// ---- DUTs/IO/Boxes/EPP2339_8DFD1558.TcDUT
{attribute 'GeneratedUsingTerminal: EPP2339-0021-0016'}
{attribute addProperty BoxType "EPP2339-0021-0016"}
{attribute addProperty Description "EPP2339-0021 16 Ch. Dig. Input/Output 24V, 0,5A, M8"}
{attribute addProperty Physics "YY"}
{attribute addProperty Id "Channel_1AT %I*Channel_830843C11Channel_2AT %I*Channel_830843C11Channel_3AT %I*Channel_830843C11Channel_4AT %I*Channel_830843C11Channel_5AT %I*Channel_830843C11Channel_6AT %I*Channel_830843C11Channel_7AT %I*Channel_830843C11Channel_8AT %I*Channel_830843C11Channel_9AT %I*Channel_830843C11Channel_10AT %I*Channel_830843C11Channel_11AT %I*Channel_830843C11Channel_12AT %I*Channel_830843C11Channel_13AT %I*Channel_830843C11Channel_14AT %I*Channel_830843C11Channel_15AT %I*Channel_830843C11Channel_16AT %I*Channel_830843C11Channel_9_1AT %Q*Channel_42CA91F71Channel_10_1AT %Q*Channel_42CA91F71Channel_11_1AT %Q*Channel_42CA91F71Channel_12_1AT %Q*Channel_42CA91F71Channel_13_1AT %Q*Channel_42CA91F71Channel_14_1AT %Q*Channel_42CA91F71Channel_15_1AT %Q*Channel_42CA91F71Channel_16_1AT %Q*Channel_42CA91F71Channel_25AT %Q*Channel_42CA91F71Channel_26AT %Q*Channel_42CA91F71Channel_27AT %Q*Channel_42CA91F71Channel_28AT %Q*Channel_42CA91F71Channel_29AT %Q*Channel_42CA91F71Channel_30AT %Q*Channel_42CA91F71Channel_31AT %Q*Channel_42CA91F71Channel_32AT %Q*Channel_42CA91F71WcStateAT %I*WcState_9091E0EB2InfoDataAT %I*InfoData_6F19DB2B2"}
{attribute addProperty CRC "2382173528"}
{attribute addProperty Size "36"}
TYPE EPP2339_8DFD1558 EXTENDS EtcSlaveBoxBase_77A0E4A7 :
STRUCT
	{attribute addProperty Name "Channel_1"}
	Channel_1 : Channel_830843C1;
	{attribute addProperty Name "Channel_2"}
	Channel_2 : Channel_830843C1;
	{attribute addProperty Name "Channel_3"}
	Channel_3 : Channel_830843C1;
	{attribute addProperty Name "Channel_4"}
	Channel_4 : Channel_830843C1;
	{attribute addProperty Name "Channel_5"}
	Channel_5 : Channel_830843C1;
	{attribute addProperty Name "Channel_6"}
	Channel_6 : Channel_830843C1;
	{attribute addProperty Name "Channel_7"}
	Channel_7 : Channel_830843C1;
	{attribute addProperty Name "Channel_8"}
	Channel_8 : Channel_830843C1;
	{attribute addProperty Name "Channel_9"}
	Channel_9 : Channel_830843C1;
	{attribute addProperty Name "Channel_10"}
	Channel_10 : Channel_830843C1;
	{attribute addProperty Name "Channel_11"}
	Channel_11 : Channel_830843C1;
	{attribute addProperty Name "Channel_12"}
	Channel_12 : Channel_830843C1;
	{attribute addProperty Name "Channel_13"}
	Channel_13 : Channel_830843C1;
	{attribute addProperty Name "Channel_14"}
	Channel_14 : Channel_830843C1;
	{attribute addProperty Name "Channel_15"}
	Channel_15 : Channel_830843C1;
	{attribute addProperty Name "Channel_16"}
	Channel_16 : Channel_830843C1;
	{attribute addProperty Name "Channel_9_1"}
	Channel_9_1 : Channel_42CA91F7;
	{attribute addProperty Name "Channel_10_1"}
	Channel_10_1 : Channel_42CA91F7;
	{attribute addProperty Name "Channel_11_1"}
	Channel_11_1 : Channel_42CA91F7;
	{attribute addProperty Name "Channel_12_1"}
	Channel_12_1 : Channel_42CA91F7;
	{attribute addProperty Name "Channel_13_1"}
	Channel_13_1 : Channel_42CA91F7;
	{attribute addProperty Name "Channel_14_1"}
	Channel_14_1 : Channel_42CA91F7;
	{attribute addProperty Name "Channel_15_1"}
	Channel_15_1 : Channel_42CA91F7;
	{attribute addProperty Name "Channel_16_1"}
	Channel_16_1 : Channel_42CA91F7;
	{attribute addProperty Name "Channel_25"}
	Channel_25 : Channel_42CA91F7;
	{attribute addProperty Name "Channel_26"}
	Channel_26 : Channel_42CA91F7;
	{attribute addProperty Name "Channel_27"}
	Channel_27 : Channel_42CA91F7;
	{attribute addProperty Name "Channel_28"}
	Channel_28 : Channel_42CA91F7;
	{attribute addProperty Name "Channel_29"}
	Channel_29 : Channel_42CA91F7;
	{attribute addProperty Name "Channel_30"}
	Channel_30 : Channel_42CA91F7;
	{attribute addProperty Name "Channel_31"}
	Channel_31 : Channel_42CA91F7;
	{attribute addProperty Name "Channel_32"}
	Channel_32 : Channel_42CA91F7;
	{attribute addProperty Name "WcState"}
	WcState : WcState_9091E0EB;
	{attribute addProperty Name "InfoData"}
	InfoData : InfoData_6F19DB2B;
END_STRUCT
END_TYPE

// ---- DUTs/IO/Boxes/EPP2349_8DFD1558.TcDUT
{attribute 'GeneratedUsingTerminal: EPP2349-0021-0016'}
{attribute addProperty BoxType "EPP2349-0021-0016"}
{attribute addProperty Description "EPP2349-0021 16 Ch. Dig. Input/Output 24V, 10µs, 0,5A, M8"}
{attribute addProperty Physics "YY"}
{attribute addProperty Id "Channel_1AT %I*Channel_830843C11Channel_2AT %I*Channel_830843C11Channel_3AT %I*Channel_830843C11Channel_4AT %I*Channel_830843C11Channel_5AT %I*Channel_830843C11Channel_6AT %I*Channel_830843C11Channel_7AT %I*Channel_830843C11Channel_8AT %I*Channel_830843C11Channel_9AT %I*Channel_830843C11Channel_10AT %I*Channel_830843C11Channel_11AT %I*Channel_830843C11Channel_12AT %I*Channel_830843C11Channel_13AT %I*Channel_830843C11Channel_14AT %I*Channel_830843C11Channel_15AT %I*Channel_830843C11Channel_16AT %I*Channel_830843C11Channel_9_1AT %Q*Channel_42CA91F71Channel_10_1AT %Q*Channel_42CA91F71Channel_11_1AT %Q*Channel_42CA91F71Channel_12_1AT %Q*Channel_42CA91F71Channel_13_1AT %Q*Channel_42CA91F71Channel_14_1AT %Q*Channel_42CA91F71Channel_15_1AT %Q*Channel_42CA91F71Channel_16_1AT %Q*Channel_42CA91F71Channel_25AT %Q*Channel_42CA91F71Channel_26AT %Q*Channel_42CA91F71Channel_27AT %Q*Channel_42CA91F71Channel_28AT %Q*Channel_42CA91F71Channel_29AT %Q*Channel_42CA91F71Channel_30AT %Q*Channel_42CA91F71Channel_31AT %Q*Channel_42CA91F71Channel_32AT %Q*Channel_42CA91F71WcStateAT %I*WcState_9091E0EB2InfoDataAT %I*InfoData_6F19DB2B2"}
{attribute addProperty CRC "2382173528"}
{attribute addProperty Size "36"}
TYPE EPP2349_8DFD1558 EXTENDS EtcSlaveBoxBase_77A0E4A7 :
STRUCT
	{attribute addProperty Name "Channel_1"}
	Channel_1 : Channel_830843C1;
	{attribute addProperty Name "Channel_2"}
	Channel_2 : Channel_830843C1;
	{attribute addProperty Name "Channel_3"}
	Channel_3 : Channel_830843C1;
	{attribute addProperty Name "Channel_4"}
	Channel_4 : Channel_830843C1;
	{attribute addProperty Name "Channel_5"}
	Channel_5 : Channel_830843C1;
	{attribute addProperty Name "Channel_6"}
	Channel_6 : Channel_830843C1;
	{attribute addProperty Name "Channel_7"}
	Channel_7 : Channel_830843C1;
	{attribute addProperty Name "Channel_8"}
	Channel_8 : Channel_830843C1;
	{attribute addProperty Name "Channel_9"}
	Channel_9 : Channel_830843C1;
	{attribute addProperty Name "Channel_10"}
	Channel_10 : Channel_830843C1;
	{attribute addProperty Name "Channel_11"}
	Channel_11 : Channel_830843C1;
	{attribute addProperty Name "Channel_12"}
	Channel_12 : Channel_830843C1;
	{attribute addProperty Name "Channel_13"}
	Channel_13 : Channel_830843C1;
	{attribute addProperty Name "Channel_14"}
	Channel_14 : Channel_830843C1;
	{attribute addProperty Name "Channel_15"}
	Channel_15 : Channel_830843C1;
	{attribute addProperty Name "Channel_16"}
	Channel_16 : Channel_830843C1;
	{attribute addProperty Name "Channel_9_1"}
	Channel_9_1 : Channel_42CA91F7;
	{attribute addProperty Name "Channel_10_1"}
	Channel_10_1 : Channel_42CA91F7;
	{attribute addProperty Name "Channel_11_1"}
	Channel_11_1 : Channel_42CA91F7;
	{attribute addProperty Name "Channel_12_1"}
	Channel_12_1 : Channel_42CA91F7;
	{attribute addProperty Name "Channel_13_1"}
	Channel_13_1 : Channel_42CA91F7;
	{attribute addProperty Name "Channel_14_1"}
	Channel_14_1 : Channel_42CA91F7;
	{attribute addProperty Name "Channel_15_1"}
	Channel_15_1 : Channel_42CA91F7;
	{attribute addProperty Name "Channel_16_1"}
	Channel_16_1 : Channel_42CA91F7;
	{attribute addProperty Name "Channel_25"}
	Channel_25 : Channel_42CA91F7;
	{attribute addProperty Name "Channel_26"}
	Channel_26 : Channel_42CA91F7;
	{attribute addProperty Name "Channel_27"}
	Channel_27 : Channel_42CA91F7;
	{attribute addProperty Name "Channel_28"}
	Channel_28 : Channel_42CA91F7;
	{attribute addProperty Name "Channel_29"}
	Channel_29 : Channel_42CA91F7;
	{attribute addProperty Name "Channel_30"}
	Channel_30 : Channel_42CA91F7;
	{attribute addProperty Name "Channel_31"}
	Channel_31 : Channel_42CA91F7;
	{attribute addProperty Name "Channel_32"}
	Channel_32 : Channel_42CA91F7;
	{attribute addProperty Name "WcState"}
	WcState : WcState_9091E0EB;
	{attribute addProperty Name "InfoData"}
	InfoData : InfoData_6F19DB2B;
END_STRUCT
END_TYPE

// ---- DUTs/IO/Boxes/EP2316_3C060514.TcDUT
{attribute 'GeneratedUsingTerminal: EP2316-0008-0017'}
{attribute addProperty BoxType "EP2316-0008-0017"}
{attribute addProperty Description "EP2316-0008 8 Ch. Dig. In, 10µs, 8Ch. Dig. Out 24V, 0,5A, Diagnostic, D-SUB25"}
{attribute addProperty Physics "YY"}
{attribute addProperty Id "DO_Diag_InputsAT %I*DO_Diag_Inputs_CC4551489DO_Diag_Inputs_1AT %I*DO_Diag_Inputs_212B82C19DO_Inputs_DeviceAT %I*DO_Inputs_Device_AF161A9E4DO_OutputsAT %Q*DO_Outputs_28AC1A9E8DO_Outputs_DeviceAT %Q*DO_Outputs_Device_36A5EF172WcStateAT %I*WcState_9091E0EB2InfoDataAT %I*InfoData_32EB74EA10"}
{attribute addProperty CRC "1007027476"}
{attribute addProperty Size "44"}
TYPE EP2316_3C060514 EXTENDS EtcSlaveBoxBase_77A0E4A7 :
STRUCT
	{attribute addProperty Name "DO_Diag_Inputs"}
	DO_Diag_Inputs : DO_Diag_Inputs_CC455148;
	{attribute addProperty Name "DO_Diag_Inputs_1"}
	DO_Diag_Inputs_1 : DO_Diag_Inputs_212B82C1;
	{attribute addProperty Name "DO_Inputs_Device"}
	DO_Inputs_Device : DO_Inputs_Device_AF161A9E;
	{attribute addProperty Name "DO_Outputs"}
	DO_Outputs : DO_Outputs_28AC1A9E;
	{attribute addProperty Name "DO_Outputs_Device"}
	DO_Outputs_Device : DO_Outputs_Device_36A5EF17;
	{attribute addProperty Name "WcState"}
	WcState : WcState_9091E0EB;
	{attribute addProperty Name "InfoData"}
	InfoData : InfoData_32EB74EA;
END_STRUCT
END_TYPE

// ---- DUTs/IO/Boxes/EP2338_39FFBC52.TcDUT
{attribute 'GeneratedUsingTerminal: EP2338-0001-0016'}
{attribute addProperty BoxType "EP2338-0001-0016"}
{attribute addProperty Description "EP2338-0001 8 Ch. Dig. Input/Output 24V, 0,5A, M8"}
{attribute addProperty Physics "YY"}
{attribute addProperty Id "Channel_1AT %I*Channel_830843C11Channel_2AT %I*Channel_830843C11Channel_3AT %I*Channel_830843C11Channel_4AT %I*Channel_830843C11Channel_5AT %I*Channel_830843C11Channel_6AT %I*Channel_830843C11Channel_7AT %I*Channel_830843C11Channel_8AT %I*Channel_830843C11Channel_1_1AT %Q*Channel_42CA91F71Channel_2_1AT %Q*Channel_42CA91F71Channel_3_1AT %Q*Channel_42CA91F71Channel_4_1AT %Q*Channel_42CA91F71Channel_5_1AT %Q*Channel_42CA91F71Channel_6_1AT %Q*Channel_42CA91F71Channel_7_1AT %Q*Channel_42CA91F71Channel_8_1AT %Q*Channel_42CA91F71WcStateAT %I*WcState_9091E0EB2InfoDataAT %I*InfoData_6F19DB2B2"}
{attribute addProperty CRC "973061202"}
{attribute addProperty Size "20"}
TYPE EP2338_39FFBC52 EXTENDS EtcSlaveBoxBase_77A0E4A7 :
STRUCT
	{attribute addProperty Name "Channel_1"}
	Channel_1 : Channel_830843C1;
	{attribute addProperty Name "Channel_2"}
	Channel_2 : Channel_830843C1;
	{attribute addProperty Name "Channel_3"}
	Channel_3 : Channel_830843C1;
	{attribute addProperty Name "Channel_4"}
	Channel_4 : Channel_830843C1;
	{attribute addProperty Name "Channel_5"}
	Channel_5 : Channel_830843C1;
	{attribute addProperty Name "Channel_6"}
	Channel_6 : Channel_830843C1;
	{attribute addProperty Name "Channel_7"}
	Channel_7 : Channel_830843C1;
	{attribute addProperty Name "Channel_8"}
	Channel_8 : Channel_830843C1;
	{attribute addProperty Name "Channel_1_1"}
	Channel_1_1 : Channel_42CA91F7;
	{attribute addProperty Name "Channel_2_1"}
	Channel_2_1 : Channel_42CA91F7;
	{attribute addProperty Name "Channel_3_1"}
	Channel_3_1 : Channel_42CA91F7;
	{attribute addProperty Name "Channel_4_1"}
	Channel_4_1 : Channel_42CA91F7;
	{attribute addProperty Name "Channel_5_1"}
	Channel_5_1 : Channel_42CA91F7;
	{attribute addProperty Name "Channel_6_1"}
	Channel_6_1 : Channel_42CA91F7;
	{attribute addProperty Name "Channel_7_1"}
	Channel_7_1 : Channel_42CA91F7;
	{attribute addProperty Name "Channel_8_1"}
	Channel_8_1 : Channel_42CA91F7;
	{attribute addProperty Name "WcState"}
	WcState : WcState_9091E0EB;
	{attribute addProperty Name "InfoData"}
	InfoData : InfoData_6F19DB2B;
END_STRUCT
END_TYPE

// ---- DUTs/IO/Boxes/EP2339_C2A6198C.TcDUT
{attribute 'GeneratedUsingTerminal: EP2339-0021-0016'}
{attribute addProperty BoxType "EP2339-0021-0016"}
{attribute addProperty Description "EP2339-0021 16 Ch. Dig. Input/Output 24V, 0,5A, M8"}
{attribute addProperty Physics "YY"}
{attribute addProperty Id "Channel_1AT %I*Channel_830843C11Channel_2AT %I*Channel_830843C11Channel_3AT %I*Channel_830843C11Channel_4AT %I*Channel_830843C11Channel_5AT %I*Channel_830843C11Channel_6AT %I*Channel_830843C11Channel_7AT %I*Channel_830843C11Channel_8AT %I*Channel_830843C11Channel_9AT %I*Channel_830843C11Channel_10AT %I*Channel_830843C11Channel_11AT %I*Channel_830843C11Channel_12AT %I*Channel_830843C11Channel_13AT %I*Channel_830843C11Channel_14AT %I*Channel_830843C11Channel_15AT %I*Channel_830843C11Channel_16AT %I*Channel_830843C11Channel_1_1AT %Q*Channel_42CA91F71Channel_2_1AT %Q*Channel_42CA91F71Channel_3_1AT %Q*Channel_42CA91F71Channel_4_1AT %Q*Channel_42CA91F71Channel_5_1AT %Q*Channel_42CA91F71Channel_6_1AT %Q*Channel_42CA91F71Channel_7_1AT %Q*Channel_42CA91F71Channel_8_1AT %Q*Channel_42CA91F71Channel_9_1AT %Q*Channel_42CA91F71Channel_10_1AT %Q*Channel_42CA91F71Channel_11_1AT %Q*Channel_42CA91F71Channel_12_1AT %Q*Channel_42CA91F71Channel_13_1AT %Q*Channel_42CA91F71Channel_14_1AT %Q*Channel_42CA91F71Channel_15_1AT %Q*Channel_42CA91F71Channel_16_1AT %Q*Channel_42CA91F71WcStateAT %I*WcState_9091E0EB2InfoDataAT %I*InfoData_0A66F0098"}
{attribute addProperty CRC "3265665420"}
{attribute addProperty Size "42"}
TYPE EP2339_C2A6198C EXTENDS EtcSlaveBoxBase_77A0E4A7 :
STRUCT
	{attribute addProperty Name "Channel_1"}
	Channel_1 : Channel_830843C1;
	{attribute addProperty Name "Channel_2"}
	Channel_2 : Channel_830843C1;
	{attribute addProperty Name "Channel_3"}
	Channel_3 : Channel_830843C1;
	{attribute addProperty Name "Channel_4"}
	Channel_4 : Channel_830843C1;
	{attribute addProperty Name "Channel_5"}
	Channel_5 : Channel_830843C1;
	{attribute addProperty Name "Channel_6"}
	Channel_6 : Channel_830843C1;
	{attribute addProperty Name "Channel_7"}
	Channel_7 : Channel_830843C1;
	{attribute addProperty Name "Channel_8"}
	Channel_8 : Channel_830843C1;
	{attribute addProperty Name "Channel_9"}
	Channel_9 : Channel_830843C1;
	{attribute addProperty Name "Channel_10"}
	Channel_10 : Channel_830843C1;
	{attribute addProperty Name "Channel_11"}
	Channel_11 : Channel_830843C1;
	{attribute addProperty Name "Channel_12"}
	Channel_12 : Channel_830843C1;
	{attribute addProperty Name "Channel_13"}
	Channel_13 : Channel_830843C1;
	{attribute addProperty Name "Channel_14"}
	Channel_14 : Channel_830843C1;
	{attribute addProperty Name "Channel_15"}
	Channel_15 : Channel_830843C1;
	{attribute addProperty Name "Channel_16"}
	Channel_16 : Channel_830843C1;
	{attribute addProperty Name "Channel_1_1"}
	Channel_1_1 : Channel_42CA91F7;
	{attribute addProperty Name "Channel_2_1"}
	Channel_2_1 : Channel_42CA91F7;
	{attribute addProperty Name "Channel_3_1"}
	Channel_3_1 : Channel_42CA91F7;
	{attribute addProperty Name "Channel_4_1"}
	Channel_4_1 : Channel_42CA91F7;
	{attribute addProperty Name "Channel_5_1"}
	Channel_5_1 : Channel_42CA91F7;
	{attribute addProperty Name "Channel_6_1"}
	Channel_6_1 : Channel_42CA91F7;
	{attribute addProperty Name "Channel_7_1"}
	Channel_7_1 : Channel_42CA91F7;
	{attribute addProperty Name "Channel_8_1"}
	Channel_8_1 : Channel_42CA91F7;
	{attribute addProperty Name "Channel_9_1"}
	Channel_9_1 : Channel_42CA91F7;
	{attribute addProperty Name "Channel_10_1"}
	Channel_10_1 : Channel_42CA91F7;
	{attribute addProperty Name "Channel_11_1"}
	Channel_11_1 : Channel_42CA91F7;
	{attribute addProperty Name "Channel_12_1"}
	Channel_12_1 : Channel_42CA91F7;
	{attribute addProperty Name "Channel_13_1"}
	Channel_13_1 : Channel_42CA91F7;
	{attribute addProperty Name "Channel_14_1"}
	Channel_14_1 : Channel_42CA91F7;
	{attribute addProperty Name "Channel_15_1"}
	Channel_15_1 : Channel_42CA91F7;
	{attribute addProperty Name "Channel_16_1"}
	Channel_16_1 : Channel_42CA91F7;
	{attribute addProperty Name "WcState"}
	WcState : WcState_9091E0EB;
	{attribute addProperty Name "InfoData"}
	InfoData : InfoData_0A66F009;
END_STRUCT
END_TYPE

// ---- DUTs/IO/Boxes/EP2339_56BCD6FB.TcDUT
{attribute 'GeneratedUsingTerminal: EP2339-0022-0016'}
{attribute addProperty BoxType "EP2339-0022-0016"}
{attribute addProperty Description "EP2339-0022 16 Ch. Dig. Input/Output 24V, 0,5A, M12"}
{attribute addProperty Physics "YY"}
{attribute addProperty Id "Channel_1AT %I*Channel_830843C11Channel_2AT %I*Channel_830843C11Channel_3AT %I*Channel_830843C11Channel_4AT %I*Channel_830843C11Channel_5AT %I*Channel_830843C11Channel_6AT %I*Channel_830843C11Channel_7AT %I*Channel_830843C11Channel_8AT %I*Channel_830843C11Channel_9AT %I*Channel_830843C11Channel_10AT %I*Channel_830843C11Channel_11AT %I*Channel_830843C11Channel_12AT %I*Channel_830843C11Channel_13AT %I*Channel_830843C11Channel_14AT %I*Channel_830843C11Channel_15AT %I*Channel_830843C11Channel_16AT %I*Channel_830843C11Channel_1_1AT %Q*Channel_42CA91F71Channel_2_1AT %Q*Channel_42CA91F71Channel_3_1AT %Q*Channel_42CA91F71Channel_4_1AT %Q*Channel_42CA91F71Channel_5_1AT %Q*Channel_42CA91F71Channel_6_1AT %Q*Channel_42CA91F71Channel_7_1AT %Q*Channel_42CA91F71Channel_8_1AT %Q*Channel_42CA91F71Channel_9_1AT %Q*Channel_42CA91F71Channel_10_1AT %Q*Channel_42CA91F71Channel_11_1AT %Q*Channel_42CA91F71Channel_12_1AT %Q*Channel_42CA91F71Channel_13_1AT %Q*Channel_42CA91F71Channel_14_1AT %Q*Channel_42CA91F71Channel_15_1AT %Q*Channel_42CA91F71Channel_16_1AT %Q*Channel_42CA91F71WcStateAT %I*WcState_9091E0EB2InfoDataAT %I*InfoData_6F19DB2B2"}
{attribute addProperty CRC "1455216379"}
{attribute addProperty Size "36"}
TYPE EP2339_56BCD6FB EXTENDS EtcSlaveBoxBase_77A0E4A7 :
STRUCT
	{attribute addProperty Name "Channel_1"}
	Channel_1 : Channel_830843C1;
	{attribute addProperty Name "Channel_2"}
	Channel_2 : Channel_830843C1;
	{attribute addProperty Name "Channel_3"}
	Channel_3 : Channel_830843C1;
	{attribute addProperty Name "Channel_4"}
	Channel_4 : Channel_830843C1;
	{attribute addProperty Name "Channel_5"}
	Channel_5 : Channel_830843C1;
	{attribute addProperty Name "Channel_6"}
	Channel_6 : Channel_830843C1;
	{attribute addProperty Name "Channel_7"}
	Channel_7 : Channel_830843C1;
	{attribute addProperty Name "Channel_8"}
	Channel_8 : Channel_830843C1;
	{attribute addProperty Name "Channel_9"}
	Channel_9 : Channel_830843C1;
	{attribute addProperty Name "Channel_10"}
	Channel_10 : Channel_830843C1;
	{attribute addProperty Name "Channel_11"}
	Channel_11 : Channel_830843C1;
	{attribute addProperty Name "Channel_12"}
	Channel_12 : Channel_830843C1;
	{attribute addProperty Name "Channel_13"}
	Channel_13 : Channel_830843C1;
	{attribute addProperty Name "Channel_14"}
	Channel_14 : Channel_830843C1;
	{attribute addProperty Name "Channel_15"}
	Channel_15 : Channel_830843C1;
	{attribute addProperty Name "Channel_16"}
	Channel_16 : Channel_830843C1;
	{attribute addProperty Name "Channel_1_1"}
	Channel_1_1 : Channel_42CA91F7;
	{attribute addProperty Name "Channel_2_1"}
	Channel_2_1 : Channel_42CA91F7;
	{attribute addProperty Name "Channel_3_1"}
	Channel_3_1 : Channel_42CA91F7;
	{attribute addProperty Name "Channel_4_1"}
	Channel_4_1 : Channel_42CA91F7;
	{attribute addProperty Name "Channel_5_1"}
	Channel_5_1 : Channel_42CA91F7;
	{attribute addProperty Name "Channel_6_1"}
	Channel_6_1 : Channel_42CA91F7;
	{attribute addProperty Name "Channel_7_1"}
	Channel_7_1 : Channel_42CA91F7;
	{attribute addProperty Name "Channel_8_1"}
	Channel_8_1 : Channel_42CA91F7;
	{attribute addProperty Name "Channel_9_1"}
	Channel_9_1 : Channel_42CA91F7;
	{attribute addProperty Name "Channel_10_1"}
	Channel_10_1 : Channel_42CA91F7;
	{attribute addProperty Name "Channel_11_1"}
	Channel_11_1 : Channel_42CA91F7;
	{attribute addProperty Name "Channel_12_1"}
	Channel_12_1 : Channel_42CA91F7;
	{attribute addProperty Name "Channel_13_1"}
	Channel_13_1 : Channel_42CA91F7;
	{attribute addProperty Name "Channel_14_1"}
	Channel_14_1 : Channel_42CA91F7;
	{attribute addProperty Name "Channel_15_1"}
	Channel_15_1 : Channel_42CA91F7;
	{attribute addProperty Name "Channel_16_1"}
	Channel_16_1 : Channel_42CA91F7;
	{attribute addProperty Name "WcState"}
	WcState : WcState_9091E0EB;
	{attribute addProperty Name "InfoData"}
	InfoData : InfoData_6F19DB2B;
END_STRUCT
END_TYPE

// ---- DUTs/IO/Boxes/EJ5151_905C5FD8.TcDUT
{attribute 'GeneratedUsingTerminal: EJ5151-0000-0016'}
{attribute addProperty BoxType "EJ5151-0000-0016"}
{attribute addProperty Description "EJ5151 1Ch. Inc. Encoder"}
{attribute addProperty Physics "KK"}
{attribute addProperty Id "ENC_InputsAT %I*ENC_Inputs_B353648514ENC_Inputs_1AT %I*ENC_Inputs_24B63C534ENC_OutputsAT %Q*ENC_Outputs_21E2D14D6WcStateAT %I*WcState_9091E0EB2InfoDataAT %I*InfoData_32EB74EA10"}
{attribute addProperty CRC "2421972952"}
{attribute addProperty Size "36"}
TYPE EJ5151_905C5FD8 EXTENDS EtcSlaveTerminalBase_947E5A46 :
STRUCT
	{attribute addProperty Name "ENC_Inputs"}
	ENC_Inputs : ENC_Inputs_B3536485;
	{attribute addProperty Name "ENC_Inputs_1"}
	ENC_Inputs_1 : ENC_Inputs_24B63C53;
	{attribute addProperty Name "ENC_Outputs"}
	ENC_Outputs : ENC_Outputs_21E2D14D;
	{attribute addProperty Name "WcState"}
	WcState : WcState_9091E0EB;
	{attribute addProperty Name "InfoData"}
	InfoData : InfoData_32EB74EA;
END_STRUCT
END_TYPE

// ---- DUTs/IO/Boxes/EL1262_0FA571DE.TcDUT
{attribute 'GeneratedUsingTerminal: EL1262-0000-0002'}
{attribute addProperty BoxType "EL1262-0000-0002"}
{attribute addProperty Description "EL1262 2Ch. Dig. Input 24V, 1µs, DC Oversample"}
{attribute addProperty Physics "KK"}
{attribute addProperty Id "Ch1_CycleCountAT %I*Ch1_CycleCount_9DBE2BC52Ch1_Input_0AT %I*Ch1_Input_FFC4CE241Ch1_Input_1AT %I*Ch1_Input_FFC4CE241Ch1_Input_2AT %I*Ch1_Input_FFC4CE241Ch1_Input_3AT %I*Ch1_Input_FFC4CE241Ch1_Input_4AT %I*Ch1_Input_FFC4CE241Ch1_Input_5AT %I*Ch1_Input_FFC4CE241Ch1_Input_6AT %I*Ch1_Input_FFC4CE241Ch1_Input_7AT %I*Ch1_Input_FFC4CE241Ch1_Input_8AT %I*Ch1_Input_FFC4CE241Ch1_Input_9AT %I*Ch1_Input_FFC4CE241GapAT %I*EMPTY_STRUCTURE0Ch2_CycleCountAT %I*Ch2_CycleCount_976A51B52Ch2_Input_0AT %I*Ch2_Input_78ADA90C1Ch2_Input_1AT %I*Ch2_Input_78ADA90C1Ch2_Input_2AT %I*Ch2_Input_78ADA90C1Ch2_Input_3AT %I*Ch2_Input_78ADA90C1Ch2_Input_4AT %I*Ch2_Input_78ADA90C1Ch2_Input_5AT %I*Ch2_Input_78ADA90C1Ch2_Input_6AT %I*Ch2_Input_78ADA90C1Ch2_Input_7AT %I*Ch2_Input_78ADA90C1Ch2_Input_8AT %I*Ch2_Input_78ADA90C1Ch2_Input_9AT %I*Ch2_Input_78ADA90C1Gap_1AT %I*EMPTY_STRUCTURE0NextSync1TimeAT %I*NextSync1Time_EE185E174WcStateAT %I*WcState_9091E0EB2InfoDataAT %I*InfoData_A7436BC610"}
{attribute addProperty CRC "262500830"}
{attribute addProperty Size "40"}
TYPE EL1262_0FA571DE EXTENDS EtcSlaveTerminalBase_947E5A46 :
STRUCT
	{attribute addProperty Name "Ch1_CycleCount"}
	Ch1_CycleCount : Ch1_CycleCount_9DBE2BC5;
	{attribute addProperty Name "Ch1_Input_0"}
	Ch1_Input_0 : Ch1_Input_FFC4CE24;
	{attribute addProperty Name "Ch1_Input_1"}
	Ch1_Input_1 : Ch1_Input_FFC4CE24;
	{attribute addProperty Name "Ch1_Input_2"}
	Ch1_Input_2 : Ch1_Input_FFC4CE24;
	{attribute addProperty Name "Ch1_Input_3"}
	Ch1_Input_3 : Ch1_Input_FFC4CE24;
	{attribute addProperty Name "Ch1_Input_4"}
	Ch1_Input_4 : Ch1_Input_FFC4CE24;
	{attribute addProperty Name "Ch1_Input_5"}
	Ch1_Input_5 : Ch1_Input_FFC4CE24;
	{attribute addProperty Name "Ch1_Input_6"}
	Ch1_Input_6 : Ch1_Input_FFC4CE24;
	{attribute addProperty Name "Ch1_Input_7"}
	Ch1_Input_7 : Ch1_Input_FFC4CE24;
	{attribute addProperty Name "Ch1_Input_8"}
	Ch1_Input_8 : Ch1_Input_FFC4CE24;
	{attribute addProperty Name "Ch1_Input_9"}
	Ch1_Input_9 : Ch1_Input_FFC4CE24;
	{attribute addProperty Name "Gap"}
	Gap : EMPTY_STRUCTURE;
	{attribute addProperty Name "Ch2_CycleCount"}
	Ch2_CycleCount : Ch2_CycleCount_976A51B5;
	{attribute addProperty Name "Ch2_Input_0"}
	Ch2_Input_0 : Ch2_Input_78ADA90C;
	{attribute addProperty Name "Ch2_Input_1"}
	Ch2_Input_1 : Ch2_Input_78ADA90C;
	{attribute addProperty Name "Ch2_Input_2"}
	Ch2_Input_2 : Ch2_Input_78ADA90C;
	{attribute addProperty Name "Ch2_Input_3"}
	Ch2_Input_3 : Ch2_Input_78ADA90C;
	{attribute addProperty Name "Ch2_Input_4"}
	Ch2_Input_4 : Ch2_Input_78ADA90C;
	{attribute addProperty Name "Ch2_Input_5"}
	Ch2_Input_5 : Ch2_Input_78ADA90C;
	{attribute addProperty Name "Ch2_Input_6"}
	Ch2_Input_6 : Ch2_Input_78ADA90C;
	{attribute addProperty Name "Ch2_Input_7"}
	Ch2_Input_7 : Ch2_Input_78ADA90C;
	{attribute addProperty Name "Ch2_Input_8"}
	Ch2_Input_8 : Ch2_Input_78ADA90C;
	{attribute addProperty Name "Ch2_Input_9"}
	Ch2_Input_9 : Ch2_Input_78ADA90C;
	{attribute addProperty Name "Gap_1"}
	Gap_1 : EMPTY_STRUCTURE;
	{attribute addProperty Name "NextSync1Time"}
	NextSync1Time : NextSync1Time_EE185E17;
	{attribute addProperty Name "WcState"}
	WcState : WcState_9091E0EB;
	{attribute addProperty Name "InfoData"}
	InfoData : InfoData_A7436BC6;
END_STRUCT
END_TYPE

// ---- DUTs/IO/Boxes/EL2262_79C970B1.TcDUT
{attribute 'GeneratedUsingTerminal: EL2262-0000-0001'}
{attribute addProperty BoxType "EL2262-0000-0001"}
{attribute addProperty Description "EL2262 2Ch. Dig. Output 24V, 0.5A, DC Over Sampling"}
{attribute addProperty Physics "KK"}
{attribute addProperty Id "CycCount0AT %Q*CycCount0_2C2338042Sample0_0AT %Q*Sample_0023574C1GapAT %I*EMPTY_STRUCTURE0CycCount1AT %Q*CycCount1_2C2338042Sample1_0AT %Q*Sample_07D5B44A1Gap_1AT %I*EMPTY_STRUCTURE0WcStateAT %I*WcState_0B2B16F91InfoDataAT %I*InfoData_A7436BC610"}
{attribute addProperty CRC "2043244721"}
{attribute addProperty Size "17"}
TYPE EL2262_79C970B1 EXTENDS EtcSlaveTerminalBase_947E5A46 :
STRUCT
	{attribute addProperty Name "CycCount0"}
	CycCount0 : CycCount0_2C233804;
	{attribute addProperty Name "Sample0_0"}
	Sample0_0 : Sample_0023574C;
	{attribute addProperty Name "Gap"}
	Gap : EMPTY_STRUCTURE;
	{attribute addProperty Name "CycCount1"}
	CycCount1 : CycCount1_2C233804;
	{attribute addProperty Name "Sample1_0"}
	Sample1_0 : Sample_07D5B44A;
	{attribute addProperty Name "Gap_1"}
	Gap_1 : EMPTY_STRUCTURE;
	{attribute addProperty Name "WcState"}
	WcState : WcState_0B2B16F9;
	{attribute addProperty Name "InfoData"}
	InfoData : InfoData_A7436BC6;
END_STRUCT
END_TYPE

// ---- DUTs/IO/Boxes/EL2262_147DB6E1.TcDUT
{attribute 'GeneratedUsingTerminal: EL2262-0000-0002'}
{attribute addProperty BoxType "EL2262-0000-0002"}
{attribute addProperty Description "EL2262 2Ch. Dig. Output 24V, 1µs, DC Oversample"}
{attribute addProperty Physics "KK"}
{attribute addProperty Id "CycCount0AT %Q*CycCount0_AF431CE02Sample0_0AT %Q*Sample_0023574C1Sample0_1AT %Q*Sample_0023574C1Sample0_2AT %Q*Sample_0023574C1Sample0_3AT %Q*Sample_0023574C1Sample0_4AT %Q*Sample_0023574C1Sample0_5AT %Q*Sample_0023574C1Sample0_6AT %Q*Sample_0023574C1Sample0_7AT %Q*Sample_0023574C1Sample0_8AT %Q*Sample_0023574C1Sample0_9AT %Q*Sample_0023574C1GapAT %I*EMPTY_STRUCTURE0CycCount1AT %Q*CycCount1_A8B5FFE62Sample1_0AT %Q*Sample_07D5B44A1Sample1_1AT %Q*Sample_07D5B44A1Sample1_2AT %Q*Sample_07D5B44A1Sample1_3AT %Q*Sample_07D5B44A1Sample1_4AT %Q*Sample_07D5B44A1Sample1_5AT %Q*Sample_07D5B44A1Sample1_6AT %Q*Sample_07D5B44A1Sample1_7AT %Q*Sample_07D5B44A1Sample1_8AT %Q*Sample_07D5B44A1Sample1_9AT %Q*Sample_07D5B44A1Gap_1AT %I*EMPTY_STRUCTURE0WcStateAT %I*WcState_0B2B16F91InfoDataAT %I*InfoData_A7436BC610"}
{attribute addProperty CRC "343783137"}
{attribute addProperty Size "35"}
TYPE EL2262_147DB6E1 EXTENDS EtcSlaveTerminalBase_947E5A46 :
STRUCT
	{attribute addProperty Name "CycCount0"}
	CycCount0 : CycCount0_AF431CE0;
	{attribute addProperty Name "Sample0_0"}
	Sample0_0 : Sample_0023574C;
	{attribute addProperty Name "Sample0_1"}
	Sample0_1 : Sample_0023574C;
	{attribute addProperty Name "Sample0_2"}
	Sample0_2 : Sample_0023574C;
	{attribute addProperty Name "Sample0_3"}
	Sample0_3 : Sample_0023574C;
	{attribute addProperty Name "Sample0_4"}
	Sample0_4 : Sample_0023574C;
	{attribute addProperty Name "Sample0_5"}
	Sample0_5 : Sample_0023574C;
	{attribute addProperty Name "Sample0_6"}
	Sample0_6 : Sample_0023574C;
	{attribute addProperty Name "Sample0_7"}
	Sample0_7 : Sample_0023574C;
	{attribute addProperty Name "Sample0_8"}
	Sample0_8 : Sample_0023574C;
	{attribute addProperty Name "Sample0_9"}
	Sample0_9 : Sample_0023574C;
	{attribute addProperty Name "Gap"}
	Gap : EMPTY_STRUCTURE;
	{attribute addProperty Name "CycCount1"}
	CycCount1 : CycCount1_A8B5FFE6;
	{attribute addProperty Name "Sample1_0"}
	Sample1_0 : Sample_07D5B44A;
	{attribute addProperty Name "Sample1_1"}
	Sample1_1 : Sample_07D5B44A;
	{attribute addProperty Name "Sample1_2"}
	Sample1_2 : Sample_07D5B44A;
	{attribute addProperty Name "Sample1_3"}
	Sample1_3 : Sample_07D5B44A;
	{attribute addProperty Name "Sample1_4"}
	Sample1_4 : Sample_07D5B44A;
	{attribute addProperty Name "Sample1_5"}
	Sample1_5 : Sample_07D5B44A;
	{attribute addProperty Name "Sample1_6"}
	Sample1_6 : Sample_07D5B44A;
	{attribute addProperty Name "Sample1_7"}
	Sample1_7 : Sample_07D5B44A;
	{attribute addProperty Name "Sample1_8"}
	Sample1_8 : Sample_07D5B44A;
	{attribute addProperty Name "Sample1_9"}
	Sample1_9 : Sample_07D5B44A;
	{attribute addProperty Name "Gap_1"}
	Gap_1 : EMPTY_STRUCTURE;
	{attribute addProperty Name "WcState"}
	WcState : WcState_0B2B16F9;
	{attribute addProperty Name "InfoData"}
	InfoData : InfoData_A7436BC6;
END_STRUCT
END_TYPE

// ---- DUTs/IO/Boxes/EL2262_9619875D.TcDUT
{attribute 'GeneratedUsingTerminal: EL2262-0000-0004'}
{attribute addProperty BoxType "EL2262-0000-0004"}
{attribute addProperty Description "EL2262 2Ch. Dig. Output 24V, 1µs, DC Oversample"}
{attribute addProperty Physics "KK"}
{attribute addProperty Id "StartTimeNextOutputAT %I*StartTimeNextOutput_228767F44CycCount0AT %Q*CycCount0_AF431CE02Sample0_0AT %Q*Sample_0023574C1Sample0_1AT %Q*Sample_0023574C1Sample0_2AT %Q*Sample_0023574C1Sample0_3AT %Q*Sample_0023574C1Sample0_4AT %Q*Sample_0023574C1Sample0_5AT %Q*Sample_0023574C1Sample0_6AT %Q*Sample_0023574C1Sample0_7AT %Q*Sample_0023574C1Sample0_8AT %Q*Sample_0023574C1Sample0_9AT %Q*Sample_0023574C1GapAT %I*EMPTY_STRUCTURE0CycCount1AT %Q*CycCount1_A8B5FFE62Sample1_0AT %Q*Sample_07D5B44A1Sample1_1AT %Q*Sample_07D5B44A1Sample1_2AT %Q*Sample_07D5B44A1Sample1_3AT %Q*Sample_07D5B44A1Sample1_4AT %Q*Sample_07D5B44A1Sample1_5AT %Q*Sample_07D5B44A1Sample1_6AT %Q*Sample_07D5B44A1Sample1_7AT %Q*Sample_07D5B44A1Sample1_8AT %Q*Sample_07D5B44A1Sample1_9AT %Q*Sample_07D5B44A1Gap_1AT %I*EMPTY_STRUCTURE0WcStateAT %I*WcState_9091E0EB2InfoDataAT %I*InfoData_A7436BC610"}
{attribute addProperty CRC "2518255453"}
{attribute addProperty Size "40"}
TYPE EL2262_9619875D EXTENDS EtcSlaveTerminalBase_947E5A46 :
STRUCT
	{attribute addProperty Name "StartTimeNextOutput"}
	StartTimeNextOutput : StartTimeNextOutput_228767F4;
	{attribute addProperty Name "CycCount0"}
	CycCount0 : CycCount0_AF431CE0;
	{attribute addProperty Name "Sample0_0"}
	Sample0_0 : Sample_0023574C;
	{attribute addProperty Name "Sample0_1"}
	Sample0_1 : Sample_0023574C;
	{attribute addProperty Name "Sample0_2"}
	Sample0_2 : Sample_0023574C;
	{attribute addProperty Name "Sample0_3"}
	Sample0_3 : Sample_0023574C;
	{attribute addProperty Name "Sample0_4"}
	Sample0_4 : Sample_0023574C;
	{attribute addProperty Name "Sample0_5"}
	Sample0_5 : Sample_0023574C;
	{attribute addProperty Name "Sample0_6"}
	Sample0_6 : Sample_0023574C;
	{attribute addProperty Name "Sample0_7"}
	Sample0_7 : Sample_0023574C;
	{attribute addProperty Name "Sample0_8"}
	Sample0_8 : Sample_0023574C;
	{attribute addProperty Name "Sample0_9"}
	Sample0_9 : Sample_0023574C;
	{attribute addProperty Name "Gap"}
	Gap : EMPTY_STRUCTURE;
	{attribute addProperty Name "CycCount1"}
	CycCount1 : CycCount1_A8B5FFE6;
	{attribute addProperty Name "Sample1_0"}
	Sample1_0 : Sample_07D5B44A;
	{attribute addProperty Name "Sample1_1"}
	Sample1_1 : Sample_07D5B44A;
	{attribute addProperty Name "Sample1_2"}
	Sample1_2 : Sample_07D5B44A;
	{attribute addProperty Name "Sample1_3"}
	Sample1_3 : Sample_07D5B44A;
	{attribute addProperty Name "Sample1_4"}
	Sample1_4 : Sample_07D5B44A;
	{attribute addProperty Name "Sample1_5"}
	Sample1_5 : Sample_07D5B44A;
	{attribute addProperty Name "Sample1_6"}
	Sample1_6 : Sample_07D5B44A;
	{attribute addProperty Name "Sample1_7"}
	Sample1_7 : Sample_07D5B44A;
	{attribute addProperty Name "Sample1_8"}
	Sample1_8 : Sample_07D5B44A;
	{attribute addProperty Name "Sample1_9"}
	Sample1_9 : Sample_07D5B44A;
	{attribute addProperty Name "Gap_1"}
	Gap_1 : EMPTY_STRUCTURE;
	{attribute addProperty Name "WcState"}
	WcState : WcState_9091E0EB;
	{attribute addProperty Name "InfoData"}
	InfoData : InfoData_A7436BC6;
END_STRUCT
END_TYPE

// ---- DUTs/IO/Boxes/EL3681_02A14E64.TcDUT
{attribute 'GeneratedUsingTerminal: EL3681-0000-0017'}
{attribute addProperty BoxType "EL3681-0000-0017"}
{attribute addProperty Description "EL3681 digital multimeter terminal"}
{attribute addProperty Physics "KK"}
{attribute addProperty Id "SAI_InputsAT %I*SAI_Inputs_3A838E1114SAI_RangeAT %I*SAI_Range_C3200E782SAI_Range_1AT %Q*SAI_Range_3710D7473WcStateAT %I*WcState_9091E0EB2InfoDataAT %I*InfoData_32EB74EA10"}
{attribute addProperty CRC "44125796"}
{attribute addProperty Size "31"}
TYPE EL3681_02A14E64 EXTENDS EtcSlaveTerminalBase_947E5A46 :
STRUCT
	{attribute addProperty Name "SAI_Inputs"}
	SAI_Inputs : SAI_Inputs_3A838E11;
	{attribute addProperty Name "SAI_Range"}
	SAI_Range : SAI_Range_C3200E78;
	{attribute addProperty Name "SAI_Range_1"}
	SAI_Range_1 : SAI_Range_3710D747;
	{attribute addProperty Name "WcState"}
	WcState : WcState_9091E0EB;
	{attribute addProperty Name "InfoData"}
	InfoData : InfoData_32EB74EA;
END_STRUCT
END_TYPE

// ---- DUTs/IO/Boxes/EL3681_0095B62C.TcDUT
{attribute 'GeneratedUsingTerminal: EL3681-0000-0018'}
{attribute addProperty BoxType "EL3681-0000-0018"}
{attribute addProperty Description "EL3681 Digital multimeter terminal"}
{attribute addProperty Physics "KK"}
{attribute addProperty Id "SAI_InputsAT %I*SAI_Inputs_84B29FE914SAI_RangeAT %I*SAI_Range_BDBF6DA92SAI_Range_1AT %Q*SAI_Range_2A187FC54WcStateAT %I*WcState_9091E0EB2InfoDataAT %I*InfoData_32EB74EA10"}
{attribute addProperty CRC "9811500"}
{attribute addProperty Size "32"}
TYPE EL3681_0095B62C EXTENDS EtcSlaveTerminalBase_947E5A46 :
STRUCT
	{attribute addProperty Name "SAI_Inputs"}
	SAI_Inputs : SAI_Inputs_84B29FE9;
	{attribute addProperty Name "SAI_Range"}
	SAI_Range : SAI_Range_BDBF6DA9;
	{attribute addProperty Name "SAI_Range_1"}
	SAI_Range_1 : SAI_Range_2A187FC5;
	{attribute addProperty Name "WcState"}
	WcState : WcState_9091E0EB;
	{attribute addProperty Name "InfoData"}
	InfoData : InfoData_32EB74EA;
END_STRUCT
END_TYPE

// ---- DUTs/IO/Boxes/EL5101_127DF9F1.TcDUT
{attribute 'GeneratedUsingTerminal: EL5101--0000'}
{attribute addProperty BoxType "EL5101--0000"}
{attribute addProperty Description "EL5101 1Ch. Encoder 5V"}
{attribute addProperty Physics "KK"}
{attribute addProperty Id "Channel_1AT %I*Channel_B90637B95Channel_1_1AT %Q*Channel_C6781B153WcStateAT %I*WcState_9091E0EB2InfoDataAT %I*InfoData_32EB74EA10"}
{attribute addProperty CRC "310245873"}
{attribute addProperty Size "20"}
TYPE EL5101_127DF9F1 EXTENDS EtcSlaveTerminalBase_947E5A46 :
STRUCT
	{attribute addProperty Name "Channel_1"}
	Channel_1 : Channel_B90637B9;
	{attribute addProperty Name "Channel_1_1"}
	Channel_1_1 : Channel_C6781B15;
	{attribute addProperty Name "WcState"}
	WcState : WcState_9091E0EB;
	{attribute addProperty Name "InfoData"}
	InfoData : InfoData_32EB74EA;
END_STRUCT
END_TYPE

// ---- DUTs/IO/Boxes/EL5151_84FDBA5C.TcDUT
{attribute 'GeneratedUsingTerminal: EL5151-0000-0016'}
{attribute addProperty BoxType "EL5151-0000-0016"}
{attribute addProperty Description "EL5151 1Ch. Inc. Encoder"}
{attribute addProperty Physics "KK"}
{attribute addProperty Id "ENC_InputsAT %I*ENC_Inputs_3399C5AA16ENC_Inputs_1AT %I*ENC_Inputs_24B63C534ENC_OutputsAT %Q*ENC_Outputs_2E45048F8WcStateAT %I*WcState_9091E0EB2InfoDataAT %I*InfoData_32EB74EA10"}
{attribute addProperty CRC "2231220828"}
{attribute addProperty Size "40"}
TYPE EL5151_84FDBA5C EXTENDS EtcSlaveTerminalBase_947E5A46 :
STRUCT
	{attribute addProperty Name "ENC_Inputs"}
	ENC_Inputs : ENC_Inputs_3399C5AA;
	{attribute addProperty Name "ENC_Inputs_1"}
	ENC_Inputs_1 : ENC_Inputs_24B63C53;
	{attribute addProperty Name "ENC_Outputs"}
	ENC_Outputs : ENC_Outputs_2E45048F;
	{attribute addProperty Name "WcState"}
	WcState : WcState_9091E0EB;
	{attribute addProperty Name "InfoData"}
	InfoData : InfoData_32EB74EA;
END_STRUCT
END_TYPE

// ---- DUTs/IO/Boxes/EL5151_93354628.TcDUT
{attribute 'GeneratedUsingTerminal: EL5151-0000-0017'}
{attribute addProperty BoxType "EL5151-0000-0017"}
{attribute addProperty Description "EL5151 1Ch. Inc. Encoder"}
{attribute addProperty Physics "KK"}
{attribute addProperty Id "ENC_InputsAT %I*ENC_Inputs_561E041F18ENC_Inputs_1AT %I*ENC_Inputs_24B63C534ENC_OutputsAT %Q*ENC_Outputs_2E45048F8WcStateAT %I*WcState_9091E0EB2InfoDataAT %I*InfoData_32EB74EA10"}
{attribute addProperty CRC "2469742120"}
{attribute addProperty Size "42"}
TYPE EL5151_93354628 EXTENDS EtcSlaveTerminalBase_947E5A46 :
STRUCT
	{attribute addProperty Name "ENC_Inputs"}
	ENC_Inputs : ENC_Inputs_561E041F;
	{attribute addProperty Name "ENC_Inputs_1"}
	ENC_Inputs_1 : ENC_Inputs_24B63C53;
	{attribute addProperty Name "ENC_Outputs"}
	ENC_Outputs : ENC_Outputs_2E45048F;
	{attribute addProperty Name "WcState"}
	WcState : WcState_9091E0EB;
	{attribute addProperty Name "InfoData"}
	InfoData : InfoData_32EB74EA;
END_STRUCT
END_TYPE

// ---- DUTs/IO/Boxes/EL5151_905C5FD8.TcDUT
{attribute 'GeneratedUsingTerminal: EL5151-0000-0020'}
{attribute addProperty BoxType "EL5151-0000-0020"}
{attribute addProperty Description "EL5151 1Ch. Inc. Encoder"}
{attribute addProperty Physics "KK"}
{attribute addProperty Id "ENC_InputsAT %I*ENC_Inputs_B353648514ENC_Inputs_1AT %I*ENC_Inputs_24B63C534ENC_OutputsAT %Q*ENC_Outputs_21E2D14D6WcStateAT %I*WcState_9091E0EB2InfoDataAT %I*InfoData_32EB74EA10"}
{attribute addProperty CRC "2421972952"}
{attribute addProperty Size "36"}
TYPE EL5151_905C5FD8 EXTENDS EtcSlaveTerminalBase_947E5A46 :
STRUCT
	{attribute addProperty Name "ENC_Inputs"}
	ENC_Inputs : ENC_Inputs_B3536485;
	{attribute addProperty Name "ENC_Inputs_1"}
	ENC_Inputs_1 : ENC_Inputs_24B63C53;
	{attribute addProperty Name "ENC_Outputs"}
	ENC_Outputs : ENC_Outputs_21E2D14D;
	{attribute addProperty Name "WcState"}
	WcState : WcState_9091E0EB;
	{attribute addProperty Name "InfoData"}
	InfoData : InfoData_32EB74EA;
END_STRUCT
END_TYPE

// ---- DUTs/IO/Boxes/EL5151_4D0E77FC.TcDUT
{attribute 'GeneratedUsingTerminal: EL5151-0080-0016'}
{attribute addProperty BoxType "EL5151-0080-0016"}
{attribute addProperty Description "EL5151-0080 1Ch. Inc. Encoder (250kHz)"}
{attribute addProperty Physics "KK"}
{attribute addProperty Id "ENC_InputsAT %I*ENC_Inputs_F139456B14ENC_Inputs_1AT %I*ENC_Inputs_24B63C534ENC_OutputsAT %Q*ENC_Outputs_6FDDC6696WcStateAT %I*WcState_9091E0EB2InfoDataAT %I*InfoData_32EB74EA10"}
{attribute addProperty CRC "1292793852"}
{attribute addProperty Size "36"}
TYPE EL5151_4D0E77FC EXTENDS EtcSlaveTerminalBase_947E5A46 :
STRUCT
	{attribute addProperty Name "ENC_Inputs"}
	ENC_Inputs : ENC_Inputs_F139456B;
	{attribute addProperty Name "ENC_Inputs_1"}
	ENC_Inputs_1 : ENC_Inputs_24B63C53;
	{attribute addProperty Name "ENC_Outputs"}
	ENC_Outputs : ENC_Outputs_6FDDC669;
	{attribute addProperty Name "WcState"}
	WcState : WcState_9091E0EB;
	{attribute addProperty Name "InfoData"}
	InfoData : InfoData_32EB74EA;
END_STRUCT
END_TYPE

// ---- DUTs/IO/Boxes/EL3773_D0D76902.TcDUT
{attribute 'GeneratedUsingTerminal: EL3773-0000-0016'}
{attribute addProperty BoxType "EL3773-0000-0016"}
{attribute addProperty Description "EL3773 3 Ch. Power Monitoring, Oversample"}
{attribute addProperty Physics "KK"}
{attribute addProperty Id "L1_Voltage_StatusAT %I*L1_Voltage_Status_784F03AD8L1_Voltage_SamplesAT %I*L1_Voltage_Samples_ED678DEE20L1_Current_SamplesAT %I*L1_Current_Samples_89E078188L1_Current_Samples_1AT %I*L1_Current_Samples_3209B12F20L2_Voltage_StatusAT %I*L2_Voltage_Status_0626A0108L2_Voltage_SamplesAT %I*L2_Voltage_Samples_D91109BE20L2_Current_StatusAT %I*L2_Current_Status_F789DBA58L2_Current_SamplesAT %I*L2_Current_Samples_067F357F20L3_Voltage_StatusAT %I*L3_Voltage_Status_2C01C17B8L3_Voltage_SamplesAT %I*L3_Voltage_Samples_CAC3758E20L3_Current_StatusAT %I*L3_Current_Status_DDAEBACE8L3_Current_SamplesAT %I*L3_Current_Samples_15AD494F20AI_Timestamp_NextSync1TimeAT %I*AI_Timestamp_NextSync1Time_9AFDC2758AI_CycleCountAT %I*AI_CycleCount_B1A935A22WcStateAT %I*WcState_9091E0EB2InfoDataAT %I*InfoData_BEF6B88E18"}
{attribute addProperty CRC "3503778050"}
{attribute addProperty Size "198"}
TYPE EL3773_D0D76902 EXTENDS EtcSlaveTerminalBase_947E5A46 :
STRUCT
	{attribute addProperty Name "L1_Voltage_Status"}
	L1_Voltage_Status : L1_Voltage_Status_784F03AD;
	{attribute addProperty Name "L1_Voltage_Samples"}
	L1_Voltage_Samples : L1_Voltage_Samples_ED678DEE;
	{attribute addProperty Name "L1_Current_Samples"}
	L1_Current_Samples : L1_Current_Samples_89E07818;
	{attribute addProperty Name "L1_Current_Samples_1"}
	L1_Current_Samples_1 : L1_Current_Samples_3209B12F;
	{attribute addProperty Name "L2_Voltage_Status"}
	L2_Voltage_Status : L2_Voltage_Status_0626A010;
	{attribute addProperty Name "L2_Voltage_Samples"}
	L2_Voltage_Samples : L2_Voltage_Samples_D91109BE;
	{attribute addProperty Name "L2_Current_Status"}
	L2_Current_Status : L2_Current_Status_F789DBA5;
	{attribute addProperty Name "L2_Current_Samples"}
	L2_Current_Samples : L2_Current_Samples_067F357F;
	{attribute addProperty Name "L3_Voltage_Status"}
	L3_Voltage_Status : L3_Voltage_Status_2C01C17B;
	{attribute addProperty Name "L3_Voltage_Samples"}
	L3_Voltage_Samples : L3_Voltage_Samples_CAC3758E;
	{attribute addProperty Name "L3_Current_Status"}
	L3_Current_Status : L3_Current_Status_DDAEBACE;
	{attribute addProperty Name "L3_Current_Samples"}
	L3_Current_Samples : L3_Current_Samples_15AD494F;
	{attribute addProperty Name "AI_Timestamp_NextSync1Time"}
	AI_Timestamp_NextSync1Time : AI_Timestamp_NextSync1Time_9AFDC275;
	{attribute addProperty Name "AI_CycleCount"}
	AI_CycleCount : AI_CycleCount_B1A935A2;
	{attribute addProperty Name "WcState"}
	WcState : WcState_9091E0EB;
	{attribute addProperty Name "InfoData"}
	InfoData : InfoData_BEF6B88E;
END_STRUCT
END_TYPE

// ---- DUTs/IO/Boxes/EM7004_866015E1.TcDUT
{attribute 'GeneratedUsingTerminal: EM7004-0000-9995'}
{attribute addProperty BoxType "EM7004-0000-9995"}
{attribute addProperty Description "EM7004 4-Axis Interface Unit"}
{attribute addProperty Physics "KK"}
{attribute addProperty Id "DigitalAT %I*Digital_BD004D6F16Encoder_Channel_1AT %I*Encoder_Channel_2E4EA2136Encoder_Channel_2AT %I*Encoder_Channel_2E4EA2136Encoder_Channel_3AT %I*Encoder_Channel_2E4EA2136Encoder_Channel_4AT %I*Encoder_Channel_2E4EA2136Digital_1AT %Q*Digital_A7E1DFAB16Analog_Channel_1AT %Q*Analog_Channel_5F9B7EA62Analog_Channel_2AT %Q*Analog_Channel_5F9B7EA62Analog_Channel_3AT %Q*Analog_Channel_5F9B7EA62Analog_Channel_4AT %Q*Analog_Channel_5F9B7EA62Encoder_Channel_1_1AT %Q*Encoder_Channel_B7999E144Encoder_Channel_2_1AT %Q*Encoder_Channel_B7999E144Encoder_Channel_3_1AT %Q*Encoder_Channel_B7999E144Encoder_Channel_4_1AT %Q*Encoder_Channel_B7999E144WcStateAT %I*WcState_9091E0EB2InfoDataAT %I*InfoData_32EB74EA10"}
{attribute addProperty CRC "2254444001"}
{attribute addProperty Size "92"}
TYPE EM7004_866015E1 EXTENDS EtcSlaveTerminalBase_947E5A46 :
STRUCT
	{attribute addProperty Name "Digital"}
	Digital : Digital_BD004D6F;
	{attribute addProperty Name "Encoder_Channel_1"}
	Encoder_Channel_1 : Encoder_Channel_2E4EA213;
	{attribute addProperty Name "Encoder_Channel_2"}
	Encoder_Channel_2 : Encoder_Channel_2E4EA213;
	{attribute addProperty Name "Encoder_Channel_3"}
	Encoder_Channel_3 : Encoder_Channel_2E4EA213;
	{attribute addProperty Name "Encoder_Channel_4"}
	Encoder_Channel_4 : Encoder_Channel_2E4EA213;
	{attribute addProperty Name "Digital_1"}
	Digital_1 : Digital_A7E1DFAB;
	{attribute addProperty Name "Analog_Channel_1"}
	Analog_Channel_1 : Analog_Channel_5F9B7EA6;
	{attribute addProperty Name "Analog_Channel_2"}
	Analog_Channel_2 : Analog_Channel_5F9B7EA6;
	{attribute addProperty Name "Analog_Channel_3"}
	Analog_Channel_3 : Analog_Channel_5F9B7EA6;
	{attribute addProperty Name "Analog_Channel_4"}
	Analog_Channel_4 : Analog_Channel_5F9B7EA6;
	{attribute addProperty Name "Encoder_Channel_1_1"}
	Encoder_Channel_1_1 : Encoder_Channel_B7999E14;
	{attribute addProperty Name "Encoder_Channel_2_1"}
	Encoder_Channel_2_1 : Encoder_Channel_B7999E14;
	{attribute addProperty Name "Encoder_Channel_3_1"}
	Encoder_Channel_3_1 : Encoder_Channel_B7999E14;
	{attribute addProperty Name "Encoder_Channel_4_1"}
	Encoder_Channel_4_1 : Encoder_Channel_B7999E14;
	{attribute addProperty Name "WcState"}
	WcState : WcState_9091E0EB;
	{attribute addProperty Name "InfoData"}
	InfoData : InfoData_32EB74EA;
END_STRUCT
END_TYPE

// ---- DUTs/IO/Boxes/AX8108_8297A621.TcDUT
{attribute 'GeneratedUsingTerminal: AX8108-0100-0101-0101'}
{attribute addProperty BoxType "AX8108-0100-0101-0101"}
{attribute addProperty Description "AX8108-0100-0101"}
{attribute addProperty Physics "KK"}
{attribute addProperty Id "DeviceDevice_6E2575772Device_SafetyDevice_Safety_C21945A160Ch_ACh_A_1FF86D8522WcStateAT %I*WcState_B516A2644InfoDataAT %I*InfoData_358A59CF25"}
{attribute addProperty CRC "2190976545"}
{attribute addProperty Size "113"}
TYPE AX8108_8297A621 EXTENDS EtcSlaveTerminalBase_947E5A46 :
STRUCT
	{attribute addProperty Name "Device"}
	Device : Device_6E257577;
	{attribute addProperty Name "Device_Safety"}
	Device_Safety : Device_Safety_C21945A1;
	{attribute addProperty Name "Ch_A"}
	Ch_A : Ch_A_1FF86D85;
	{attribute addProperty Name "WcState"}
	WcState : WcState_B516A264;
	{attribute addProperty Name "InfoData"}
	InfoData : InfoData_358A59CF;
END_STRUCT
END_TYPE

// ---- DUTs/IO/Boxes/AX8108_F7A82895.TcDUT
{attribute 'GeneratedUsingTerminal: AX8108-0100-0102-0102'}
{attribute addProperty BoxType "AX8108-0100-0102-0102"}
{attribute addProperty Description "AX8108-0100-0102"}
{attribute addProperty Physics "KK"}
{attribute addProperty Id "DeviceDevice_6E2575772Device_SafetyDevice_Safety_C21945A160Ch_ACh_A_D18C6F1622WcStateAT %I*WcState_B516A2644InfoDataAT %I*InfoData_358A59CF25"}
{attribute addProperty CRC "4154992789"}
{attribute addProperty Size "113"}
TYPE AX8108_F7A82895 EXTENDS EtcSlaveTerminalBase_947E5A46 :
STRUCT
	{attribute addProperty Name "Device"}
	Device : Device_6E257577;
	{attribute addProperty Name "Device_Safety"}
	Device_Safety : Device_Safety_C21945A1;
	{attribute addProperty Name "Ch_A"}
	Ch_A : Ch_A_D18C6F16;
	{attribute addProperty Name "WcState"}
	WcState : WcState_B516A264;
	{attribute addProperty Name "InfoData"}
	InfoData : InfoData_358A59CF;
END_STRUCT
END_TYPE

// ---- DUTs/IO/Boxes/AX8118_8297A621.TcDUT
{attribute 'GeneratedUsingTerminal: AX8118-0100-0101-0101'}
{attribute addProperty BoxType "AX8118-0100-0101-0101"}
{attribute addProperty Description "AX8118-0100-0101"}
{attribute addProperty Physics "KK"}
{attribute addProperty Id "DeviceDevice_6E2575772Device_SafetyDevice_Safety_C21945A160Ch_ACh_A_1FF86D8522WcStateAT %I*WcState_B516A2644InfoDataAT %I*InfoData_358A59CF25"}
{attribute addProperty CRC "2190976545"}
{attribute addProperty Size "113"}
TYPE AX8118_8297A621 EXTENDS EtcSlaveTerminalBase_947E5A46 :
STRUCT
	{attribute addProperty Name "Device"}
	Device : Device_6E257577;
	{attribute addProperty Name "Device_Safety"}
	Device_Safety : Device_Safety_C21945A1;
	{attribute addProperty Name "Ch_A"}
	Ch_A : Ch_A_1FF86D85;
	{attribute addProperty Name "WcState"}
	WcState : WcState_B516A264;
	{attribute addProperty Name "InfoData"}
	InfoData : InfoData_358A59CF;
END_STRUCT
END_TYPE

// ---- DUTs/IO/Boxes/AX8118_F7A82895.TcDUT
{attribute 'GeneratedUsingTerminal: AX8118-0100-0102-0102'}
{attribute addProperty BoxType "AX8118-0100-0102-0102"}
{attribute addProperty Description "AX8118-0100-0102"}
{attribute addProperty Physics "KK"}
{attribute addProperty Id "DeviceDevice_6E2575772Device_SafetyDevice_Safety_C21945A160Ch_ACh_A_D18C6F1622WcStateAT %I*WcState_B516A2644InfoDataAT %I*InfoData_358A59CF25"}
{attribute addProperty CRC "4154992789"}
{attribute addProperty Size "113"}
TYPE AX8118_F7A82895 EXTENDS EtcSlaveTerminalBase_947E5A46 :
STRUCT
	{attribute addProperty Name "Device"}
	Device : Device_6E257577;
	{attribute addProperty Name "Device_Safety"}
	Device_Safety : Device_Safety_C21945A1;
	{attribute addProperty Name "Ch_A"}
	Ch_A : Ch_A_D18C6F16;
	{attribute addProperty Name "WcState"}
	WcState : WcState_B516A264;
	{attribute addProperty Name "InfoData"}
	InfoData : InfoData_358A59CF;
END_STRUCT
END_TYPE

// ---- DUTs/IO/Boxes/AX8206_63F473B4.TcDUT
{attribute 'GeneratedUsingTerminal: AX8206-0100-0101-0101'}
{attribute addProperty BoxType "AX8206-0100-0101-0101"}
{attribute addProperty Description "AX8206-0100-0101"}
{attribute addProperty Physics "KK"}
{attribute addProperty Id "DeviceDevice_6E2575772Device_SafetyDevice_Safety_C21945A160Ch_ACh_A_1FF86D8522Ch_BCh_B_5E084BAA22WcStateAT %I*WcState_B516A2644InfoDataAT %I*InfoData_386C00A526"}
{attribute addProperty CRC "1676964788"}
{attribute addProperty Size "136"}
TYPE AX8206_63F473B4 EXTENDS EtcSlaveTerminalBase_947E5A46 :
STRUCT
	{attribute addProperty Name "Device"}
	Device : Device_6E257577;
	{attribute addProperty Name "Device_Safety"}
	Device_Safety : Device_Safety_C21945A1;
	{attribute addProperty Name "Ch_A"}
	Ch_A : Ch_A_1FF86D85;
	{attribute addProperty Name "Ch_B"}
	Ch_B : Ch_B_5E084BAA;
	{attribute addProperty Name "WcState"}
	WcState : WcState_B516A264;
	{attribute addProperty Name "InfoData"}
	InfoData : InfoData_386C00A5;
END_STRUCT
END_TYPE

// ---- DUTs/IO/Boxes/AX8206_FA9FF81E.TcDUT
{attribute 'GeneratedUsingTerminal: AX8206-0100-0102-0102'}
{attribute addProperty BoxType "AX8206-0100-0102-0102"}
{attribute addProperty Description "AX8206-0100-0102"}
{attribute addProperty Physics "KK"}
{attribute addProperty Id "DeviceDevice_6E2575772Device_SafetyDevice_Safety_C21945A160Ch_ACh_A_D18C6F1622Ch_BCh_B_647F9A0C22WcStateAT %I*WcState_B516A2644InfoDataAT %I*InfoData_386C00A526"}
{attribute addProperty CRC "4204787742"}
{attribute addProperty Size "136"}
TYPE AX8206_FA9FF81E EXTENDS EtcSlaveTerminalBase_947E5A46 :
STRUCT
	{attribute addProperty Name "Device"}
	Device : Device_6E257577;
	{attribute addProperty Name "Device_Safety"}
	Device_Safety : Device_Safety_C21945A1;
	{attribute addProperty Name "Ch_A"}
	Ch_A : Ch_A_D18C6F16;
	{attribute addProperty Name "Ch_B"}
	Ch_B : Ch_B_647F9A0C;
	{attribute addProperty Name "WcState"}
	WcState : WcState_B516A264;
	{attribute addProperty Name "InfoData"}
	InfoData : InfoData_386C00A5;
END_STRUCT
END_TYPE

// ---- DUTs/IO/Boxes/AMP8000_F7A82895.TcDUT
{attribute 'GeneratedUsingTerminal: AMP8000-0030-0103-0103'}
{attribute addProperty BoxType "AMP8000-0030-0103-0103"}
{attribute addProperty Description "AMP8000-0030-0103"}
{attribute addProperty Physics "Y"}
{attribute addProperty Id "DeviceDevice_6E2575772Device_SafetyDevice_Safety_C21945A160Ch_ACh_A_D18C6F1622WcStateAT %I*WcState_B516A2644InfoDataAT %I*InfoData_358A59CF25"}
{attribute addProperty CRC "4154992789"}
{attribute addProperty Size "113"}
TYPE AMP8000_F7A82895 EXTENDS EtcSlaveBoxBase_77A0E4A7 :
STRUCT
	{attribute addProperty Name "Device"}
	Device : Device_6E257577;
	{attribute addProperty Name "Device_Safety"}
	Device_Safety : Device_Safety_C21945A1;
	{attribute addProperty Name "Ch_A"}
	Ch_A : Ch_A_D18C6F16;
	{attribute addProperty Name "WcState"}
	WcState : WcState_B516A264;
	{attribute addProperty Name "InfoData"}
	InfoData : InfoData_358A59CF;
END_STRUCT
END_TYPE

// ---- DUTs/IO/Devices/SyncUnitTask_2D604ED5.TcDUT
{attribute 'GeneratedUsingTerminal: IODEVICETYPE_ETHERCATPROT'}
{attribute addProperty BoxType "IODEVICETYPE_ETHERCATPROT"}
{attribute addProperty Id "WcStateAT %I*WcState_0B2B16F91InfoDataAT %I*InfoData_2A97D6CF8"}
{attribute addProperty CRC "761286357"}
{attribute addProperty Size "9"}
TYPE SyncUnitTask_2D604ED5 :
STRUCT
	{attribute addProperty Name "WcState"}
	WcState : WcState_0B2B16F9;
	{attribute addProperty Name "InfoData"}
	InfoData : InfoData_2A97D6CF;
END_STRUCT
END_TYPE

// ---- DUTs/IO/Devices/SyncUnitTasks_6FEB8257.TcDUT
{attribute 'GeneratedUsingTerminal: '}
{attribute addProperty BoxType ""}
{attribute addProperty Id "unreferencedAT %I*SyncUnitTask_2D604ED59PlcTaskAT %I*SyncUnitTask_2D604ED59"}
{attribute addProperty CRC "1877705303"}
{attribute addProperty Size "18"}
TYPE SyncUnitTasks_6FEB8257 :
STRUCT
	{attribute addProperty Name "unreferenced"}
	unreferenced : SyncUnitTask_2D604ED5;
	{attribute addProperty Name "PlcTask"}
	PlcTask : SyncUnitTask_2D604ED5;
END_STRUCT
END_TYPE

// ---- DUTs/IO/Devices/SyncUnits_99E584AF.TcDUT
{attribute 'GeneratedUsingTerminal: '}
{attribute addProperty BoxType ""}
{attribute addProperty Id "_defaultAT %I*SyncUnitTasks_6FEB825718"}
{attribute addProperty CRC "2581955759"}
{attribute addProperty Size "18"}
TYPE SyncUnits_99E584AF :
STRUCT
	{attribute addProperty Name "_default"}
	_default : SyncUnitTasks_6FEB8257;
END_STRUCT
END_TYPE

// ---- DUTs/IO/Topology/boxesEK1122_B55A8AA2.TcDUT
{attribute 'GeneratedUsingTerminal: EK1122-0000-0018'}
{attribute addProperty BoxType "EK1122-0000-0018"}
{attribute addProperty Id "boxessub_EK1100EK1100_1FC0878B2A_0030_EPP2339_0021_0016EPP2339_8DFD155836A_0031_EPP2339_0022_0016EPP2339_8DFD155836A_0032_EPP2349_0021_0016EPP2349_8DFD155836A_0033_EPP2349_0022_0016EPP2349_8DFD155836A_0034_EP2316_0008_0017EP2316_3C06051444A_0035_EP2338_0001_0016EP2338_39FFBC5220A_0036_EP2338_0001_0017EP2338_39FFBC5220A_0037_EP2338_0002_0016EP2338_39FFBC5220A_0038_EP2338_0002_0017EP2338_39FFBC5220A_0039_EP2339_0021_0016EP2339_C2A6198C42A_0040_EP2339_0022_0016EP2339_56BCD6FB36"}
{attribute addProperty CRC "3042609826"}
{attribute addProperty Size "348"}
{attribute addProperty Name "boxesEK1122"}
TYPE boxesEK1122_B55A8AA2 EXTENDS EK1122_1FC0878B :
STRUCT
	{attribute addProperty Name "boxessub EK1100"}
	{attribute addProperty PreviousPort "boxesEK1122 : D"}
	boxessub_EK1100 : EK1100_1FC0878B;
	{attribute addProperty Name "A_0030(EPP2339-0021-0016 )"}
	{attribute addProperty PreviousPort "boxessub EK1100 : C"}
	A_0030_EPP2339_0021_0016 : EPP2339_8DFD1558;
	{attribute addProperty Name "A_0031(EPP2339-0022-0016 )"}
	{attribute addProperty PreviousPort "A_0030(EPP2339-0021-0016 ) : B"}
	A_0031_EPP2339_0022_0016 : EPP2339_8DFD1558;
	{attribute addProperty Name "A_0032(EPP2349-0021-0016 )"}
	{attribute addProperty PreviousPort "A_0031(EPP2339-0022-0016 ) : B"}
	A_0032_EPP2349_0021_0016 : EPP2349_8DFD1558;
	{attribute addProperty Name "A_0033(EPP2349-0022-0016 )"}
	{attribute addProperty PreviousPort "A_0032(EPP2349-0021-0016 ) : B"}
	A_0033_EPP2349_0022_0016 : EPP2349_8DFD1558;
	{attribute addProperty Name "A_0034(EP2316-0008-0017 )"}
	{attribute addProperty PreviousPort "A_0033(EPP2349-0022-0016 ) : B"}
	A_0034_EP2316_0008_0017 : EP2316_3C060514;
	{attribute addProperty Name "A_0035(EP2338-0001-0016 )"}
	{attribute addProperty PreviousPort "A_0034(EP2316-0008-0017 ) : B"}
	A_0035_EP2338_0001_0016 : EP2338_39FFBC52;
	{attribute addProperty Name "A_0036(EP2338-0001-0017 )"}
	{attribute addProperty PreviousPort "A_0035(EP2338-0001-0016 ) : B"}
	A_0036_EP2338_0001_0017 : EP2338_39FFBC52;
	{attribute addProperty Name "A_0037(EP2338-0002-0016 )"}
	{attribute addProperty PreviousPort "A_0036(EP2338-0001-0017 ) : B"}
	A_0037_EP2338_0002_0016 : EP2338_39FFBC52;
	{attribute addProperty Name "A_0038(EP2338-0002-0017 )"}
	{attribute addProperty PreviousPort "A_0037(EP2338-0002-0016 ) : B"}
	A_0038_EP2338_0002_0017 : EP2338_39FFBC52;
	{attribute addProperty Name "A_0039(EP2339-0021-0016 )"}
	{attribute addProperty PreviousPort "A_0038(EP2338-0002-0017 ) : B"}
	A_0039_EP2339_0021_0016 : EP2339_C2A6198C;
	{attribute addProperty Name "A_0040(EP2339-0022-0016 )"}
	{attribute addProperty PreviousPort "A_0039(EP2339-0021-0016 ) : B"}
	A_0040_EP2339_0022_0016 : EP2339_56BCD6FB;
END_STRUCT
END_TYPE

// ---- DUTs/IO/Topology/boxes_17897972.TcDUT
{attribute 'GeneratedUsingTerminal: EK1100-0000-0018'}
{attribute addProperty BoxType "EK1100-0000-0018"}
{attribute addProperty Id "boxesEK1122boxesEK1122_B55A8AA2348A_0001_EJ5151_0000_0016EJ5151_905C5FD836A_0002_EL1262_0000_0002EL1262_0FA571DE40A_0003_EL1262_0000_0003EL1262_0FA571DE40A_0004_EL1262_0050_0002EL1262_0FA571DE40A_0005_EL1262_0050_0003EL1262_0FA571DE40A_0006_EL2262_0000_0001EL2262_79C970B117A_0007_EL2262_0000_0002EL2262_147DB6E135A_0008_EL2262_0000_0003EL2262_147DB6E135A_0009_EL2262_0000_0004EL2262_9619875D40A_0010_EL3681_0000_0017EL3681_02A14E6431A_0011_EL3681_0000_0018EL3681_0095B62C32A_0012_EL3681_0000_0019EL3681_0095B62C32A_0013_EL3681_0000_0020EL3681_0095B62C32A_0014_EL5101_0000_0000EL5101_127DF9F120A_0015_EL5151_0000_0016EL5151_84FDBA5C40A_0016_EL5151_0000_0017EL5151_9335462842A_0017_EL5151_0000_0018EL5151_9335462842A_0018_EL5151_0000_0019EL5151_9335462842A_0019_EL5151_0000_0020EL5151_905C5FD836A_0020_EL5151_0000_0025EL5151_905C5FD836A_0021_EL5151_0000_0026EL5151_905C5FD836A_0022_EL5151_0080_0016EL5151_4D0E77FC36A_0023_EL5151_0080_0017EL5151_905C5FD836A_0024_EL5151_0080_0018EL5151_905C5FD836A_0025_EL5151_0080_0019EL5151_905C5FD836A_0026_EL5151_0080_0020EL5151_905C5FD836A_0027_EL5151_0080_0021EL5151_905C5FD836A_0028_EL3773_0000_0016EL3773_D0D76902198A_0029_EM7004_0000_9995EM7004_866015E192A_0041_AX8108_0100_0101AX8108_8297A621113A_0042_AX8108_0100_0102AX8108_F7A82895113A_0043_AX8108_0100_0103AX8108_F7A82895113A_0044_AX8108_0100_0104AX8108_F7A82895113A_0045_AX8108_0110_0102AX8108_F7A82895113A_0046_AX8108_0110_0103AX8108_F7A82895113A_0047_AX8108_0110_0104AX8108_F7A82895113A_0048_AX8108_0200_0103AX8108_F7A82895113A_0049_AX8108_0200_0104AX8108_F7A82895113A_0050_AX8108_0210_0103AX8108_F7A82895113A_0051_AX8108_0210_0104AX8108_F7A82895113A_0052_AX8118_0100_0101AX8118_8297A621113A_0053_AX8118_0100_0102AX8118_F7A82895113A_0054_AX8118_0100_0103AX8118_F7A82895113A_0055_AX8118_0100_0104AX8118_F7A82895113A_0056_AX8118_0110_0102AX8118_F7A82895113A_0057_AX8118_0110_0103AX8118_F7A82895113A_0058_AX8118_0110_0104AX8118_F7A82895113A_0059_AX8118_0200_0103AX8118_F7A82895113A_0060_AX8118_0200_0104AX8118_F7A82895113A_0061_AX8118_0210_0103AX8118_F7A82895113A_0062_AX8118_0210_0104AX8118_F7A82895113A_0063_AX8206_0100_0101AX8206_63F473B4136A_0064_AX8206_0100_0102AX8206_FA9FF81E136A_0065_AX8206_0100_0103AX8206_FA9FF81E136A_0066_AX8206_0100_0104AX8206_FA9FF81E136A_0067_AX8206_0110_0102AX8206_FA9FF81E136A_0068_AX8206_0110_0103AX8206_FA9FF81E136A_0069_AX8206_0110_0104AX8206_FA9FF81E136A_0070_AX8206_0200_0103AX8206_FA9FF81E136A_0071_AX8206_0200_0104AX8206_FA9FF81E136A_0072_AX8206_0210_0103AX8206_FA9FF81E136A_0073_AX8206_0210_0104AX8206_FA9FF81E136A_0074_EM7004_0000_9995EM7004_866015E192A_0075_AX8118_0100_0101AX8118_8297A621113"}
{attribute addProperty CRC "394885490"}
{attribute addProperty Size "5785"}
{attribute addProperty Name "boxes"}
TYPE boxes_17897972 EXTENDS EK1100_1FC0878B :
STRUCT
	{attribute addProperty Name "boxesEK1122"}
	{attribute addProperty PreviousPort "boxes : B"}
	boxesEK1122 : boxesEK1122_B55A8AA2;
	{attribute addProperty Name "A_0001(EJ5151-0000-0016 )"}
	{attribute addProperty PreviousPort "boxesEK1122 : C"}
	A_0001_EJ5151_0000_0016 : EJ5151_905C5FD8;
	{attribute addProperty Name "A_0002(EL1262-0000-0002 )"}
	{attribute addProperty PreviousPort "A_0001(EJ5151-0000-0016 ) : B"}
	A_0002_EL1262_0000_0002 : EL1262_0FA571DE;
	{attribute addProperty Name "A_0003(EL1262-0000-0003 )"}
	{attribute addProperty PreviousPort "A_0002(EL1262-0000-0002 ) : B"}
	A_0003_EL1262_0000_0003 : EL1262_0FA571DE;
	{attribute addProperty Name "A_0004(EL1262-0050-0002 )"}
	{attribute addProperty PreviousPort "A_0003(EL1262-0000-0003 ) : B"}
	A_0004_EL1262_0050_0002 : EL1262_0FA571DE;
	{attribute addProperty Name "A_0005(EL1262-0050-0003 )"}
	{attribute addProperty PreviousPort "A_0004(EL1262-0050-0002 ) : B"}
	A_0005_EL1262_0050_0003 : EL1262_0FA571DE;
	{attribute addProperty Name "A_0006(EL2262-0000-0001 )"}
	{attribute addProperty PreviousPort "A_0005(EL1262-0050-0003 ) : B"}
	A_0006_EL2262_0000_0001 : EL2262_79C970B1;
	{attribute addProperty Name "A_0007(EL2262-0000-0002 )"}
	{attribute addProperty PreviousPort "A_0006(EL2262-0000-0001 ) : B"}
	A_0007_EL2262_0000_0002 : EL2262_147DB6E1;
	{attribute addProperty Name "A_0008(EL2262-0000-0003 )"}
	{attribute addProperty PreviousPort "A_0007(EL2262-0000-0002 ) : B"}
	A_0008_EL2262_0000_0003 : EL2262_147DB6E1;
	{attribute addProperty Name "A_0009(EL2262-0000-0004 )"}
	{attribute addProperty PreviousPort "A_0008(EL2262-0000-0003 ) : B"}
	A_0009_EL2262_0000_0004 : EL2262_9619875D;
	{attribute addProperty Name "A_0010(EL3681-0000-0017 )"}
	{attribute addProperty PreviousPort "A_0009(EL2262-0000-0004 ) : B"}
	A_0010_EL3681_0000_0017 : EL3681_02A14E64;
	{attribute addProperty Name "A_0011(EL3681-0000-0018 )"}
	{attribute addProperty PreviousPort "A_0010(EL3681-0000-0017 ) : B"}
	A_0011_EL3681_0000_0018 : EL3681_0095B62C;
	{attribute addProperty Name "A_0012(EL3681-0000-0019 )"}
	{attribute addProperty PreviousPort "A_0011(EL3681-0000-0018 ) : B"}
	A_0012_EL3681_0000_0019 : EL3681_0095B62C;
	{attribute addProperty Name "A_0013(EL3681-0000-0020 )"}
	{attribute addProperty PreviousPort "A_0012(EL3681-0000-0019 ) : B"}
	A_0013_EL3681_0000_0020 : EL3681_0095B62C;
	{attribute addProperty Name "A_0014(EL5101-0000-0000 )"}
	{attribute addProperty PreviousPort "A_0013(EL3681-0000-0020 ) : B"}
	A_0014_EL5101_0000_0000 : EL5101_127DF9F1;
	{attribute addProperty Name "A_0015(EL5151-0000-0016 )"}
	{attribute addProperty PreviousPort "A_0014(EL5101-0000-0000 ) : B"}
	A_0015_EL5151_0000_0016 : EL5151_84FDBA5C;
	{attribute addProperty Name "A_0016(EL5151-0000-0017 )"}
	{attribute addProperty PreviousPort "A_0015(EL5151-0000-0016 ) : B"}
	A_0016_EL5151_0000_0017 : EL5151_93354628;
	{attribute addProperty Name "A_0017(EL5151-0000-0018 )"}
	{attribute addProperty PreviousPort "A_0016(EL5151-0000-0017 ) : B"}
	A_0017_EL5151_0000_0018 : EL5151_93354628;
	{attribute addProperty Name "A_0018(EL5151-0000-0019 )"}
	{attribute addProperty PreviousPort "A_0017(EL5151-0000-0018 ) : B"}
	A_0018_EL5151_0000_0019 : EL5151_93354628;
	{attribute addProperty Name "A_0019(EL5151-0000-0020 )"}
	{attribute addProperty PreviousPort "A_0018(EL5151-0000-0019 ) : B"}
	A_0019_EL5151_0000_0020 : EL5151_905C5FD8;
	{attribute addProperty Name "A_0020(EL5151-0000-0025 )"}
	{attribute addProperty PreviousPort "A_0019(EL5151-0000-0020 ) : B"}
	A_0020_EL5151_0000_0025 : EL5151_905C5FD8;
	{attribute addProperty Name "A_0021(EL5151-0000-0026 )"}
	{attribute addProperty PreviousPort "A_0020(EL5151-0000-0025 ) : B"}
	A_0021_EL5151_0000_0026 : EL5151_905C5FD8;
	{attribute addProperty Name "A_0022(EL5151-0080-0016 )"}
	{attribute addProperty PreviousPort "A_0021(EL5151-0000-0026 ) : B"}
	A_0022_EL5151_0080_0016 : EL5151_4D0E77FC;
	{attribute addProperty Name "A_0023(EL5151-0080-0017 )"}
	{attribute addProperty PreviousPort "A_0022(EL5151-0080-0016 ) : B"}
	A_0023_EL5151_0080_0017 : EL5151_905C5FD8;
	{attribute addProperty Name "A_0024(EL5151-0080-0018 )"}
	{attribute addProperty PreviousPort "A_0023(EL5151-0080-0017 ) : B"}
	A_0024_EL5151_0080_0018 : EL5151_905C5FD8;
	{attribute addProperty Name "A_0025(EL5151-0080-0019 )"}
	{attribute addProperty PreviousPort "A_0024(EL5151-0080-0018 ) : B"}
	A_0025_EL5151_0080_0019 : EL5151_905C5FD8;
	{attribute addProperty Name "A_0026(EL5151-0080-0020 )"}
	{attribute addProperty PreviousPort "A_0025(EL5151-0080-0019 ) : B"}
	A_0026_EL5151_0080_0020 : EL5151_905C5FD8;
	{attribute addProperty Name "A_0027(EL5151-0080-0021 )"}
	{attribute addProperty PreviousPort "A_0026(EL5151-0080-0020 ) : B"}
	A_0027_EL5151_0080_0021 : EL5151_905C5FD8;
	{attribute addProperty Name "A_0028(EL3773-0000-0016 )"}
	{attribute addProperty PreviousPort "A_0027(EL5151-0080-0021 ) : B"}
	A_0028_EL3773_0000_0016 : EL3773_D0D76902;
	{attribute addProperty Name "A_0029(EM7004-0000-9995 )"}
	{attribute addProperty PreviousPort "A_0028(EL3773-0000-0016 ) : B"}
	A_0029_EM7004_0000_9995 : EM7004_866015E1;
	{attribute addProperty Name "A_0041(AX8108-0100-0101 )"}
	{attribute addProperty PreviousPort "A_0029(EM7004-0000-9995 ) : B"}
	A_0041_AX8108_0100_0101 : AX8108_8297A621;
	{attribute addProperty Name "A_0042(AX8108-0100-0102 )"}
	{attribute addProperty PreviousPort "A_0041(AX8108-0100-0101 ) : B"}
	A_0042_AX8108_0100_0102 : AX8108_F7A82895;
	{attribute addProperty Name "A_0043(AX8108-0100-0103 )"}
	{attribute addProperty PreviousPort "A_0042(AX8108-0100-0102 ) : B"}
	A_0043_AX8108_0100_0103 : AX8108_F7A82895;
	{attribute addProperty Name "A_0044(AX8108-0100-0104 )"}
	{attribute addProperty PreviousPort "A_0043(AX8108-0100-0103 ) : B"}
	A_0044_AX8108_0100_0104 : AX8108_F7A82895;
	{attribute addProperty Name "A_0045(AX8108-0110-0102 )"}
	{attribute addProperty PreviousPort "A_0044(AX8108-0100-0104 ) : B"}
	A_0045_AX8108_0110_0102 : AX8108_F7A82895;
	{attribute addProperty Name "A_0046(AX8108-0110-0103 )"}
	{attribute addProperty PreviousPort "A_0045(AX8108-0110-0102 ) : B"}
	A_0046_AX8108_0110_0103 : AX8108_F7A82895;
	{attribute addProperty Name "A_0047(AX8108-0110-0104 )"}
	{attribute addProperty PreviousPort "A_0046(AX8108-0110-0103 ) : B"}
	A_0047_AX8108_0110_0104 : AX8108_F7A82895;
	{attribute addProperty Name "A_0048(AX8108-0200-0103 )"}
	{attribute addProperty PreviousPort "A_0047(AX8108-0110-0104 ) : B"}
	A_0048_AX8108_0200_0103 : AX8108_F7A82895;
	{attribute addProperty Name "A_0049(AX8108-0200-0104 )"}
	{attribute addProperty PreviousPort "A_0048(AX8108-0200-0103 ) : B"}
	A_0049_AX8108_0200_0104 : AX8108_F7A82895;
	{attribute addProperty Name "A_0050(AX8108-0210-0103 )"}
	{attribute addProperty PreviousPort "A_0049(AX8108-0200-0104 ) : B"}
	A_0050_AX8108_0210_0103 : AX8108_F7A82895;
	{attribute addProperty Name "A_0051(AX8108-0210-0104 )"}
	{attribute addProperty PreviousPort "A_0050(AX8108-0210-0103 ) : B"}
	A_0051_AX8108_0210_0104 : AX8108_F7A82895;
	{attribute addProperty Name "A_0052(AX8118-0100-0101 )"}
	{attribute addProperty PreviousPort "A_0051(AX8108-0210-0104 ) : B"}
	A_0052_AX8118_0100_0101 : AX8118_8297A621;
	{attribute addProperty Name "A_0053(AX8118-0100-0102 )"}
	{attribute addProperty PreviousPort "A_0052(AX8118-0100-0101 ) : B"}
	A_0053_AX8118_0100_0102 : AX8118_F7A82895;
	{attribute addProperty Name "A_0054(AX8118-0100-0103 )"}
	{attribute addProperty PreviousPort "A_0053(AX8118-0100-0102 ) : B"}
	A_0054_AX8118_0100_0103 : AX8118_F7A82895;
	{attribute addProperty Name "A_0055(AX8118-0100-0104 )"}
	{attribute addProperty PreviousPort "A_0054(AX8118-0100-0103 ) : B"}
	A_0055_AX8118_0100_0104 : AX8118_F7A82895;
	{attribute addProperty Name "A_0056(AX8118-0110-0102 )"}
	{attribute addProperty PreviousPort "A_0055(AX8118-0100-0104 ) : B"}
	A_0056_AX8118_0110_0102 : AX8118_F7A82895;
	{attribute addProperty Name "A_0057(AX8118-0110-0103 )"}
	{attribute addProperty PreviousPort "A_0056(AX8118-0110-0102 ) : B"}
	A_0057_AX8118_0110_0103 : AX8118_F7A82895;
	{attribute addProperty Name "A_0058(AX8118-0110-0104 )"}
	{attribute addProperty PreviousPort "A_0057(AX8118-0110-0103 ) : B"}
	A_0058_AX8118_0110_0104 : AX8118_F7A82895;
	{attribute addProperty Name "A_0059(AX8118-0200-0103 )"}
	{attribute addProperty PreviousPort "A_0058(AX8118-0110-0104 ) : B"}
	A_0059_AX8118_0200_0103 : AX8118_F7A82895;
	{attribute addProperty Name "A_0060(AX8118-0200-0104 )"}
	{attribute addProperty PreviousPort "A_0059(AX8118-0200-0103 ) : B"}
	A_0060_AX8118_0200_0104 : AX8118_F7A82895;
	{attribute addProperty Name "A_0061(AX8118-0210-0103 )"}
	{attribute addProperty PreviousPort "A_0060(AX8118-0200-0104 ) : B"}
	A_0061_AX8118_0210_0103 : AX8118_F7A82895;
	{attribute addProperty Name "A_0062(AX8118-0210-0104 )"}
	{attribute addProperty PreviousPort "A_0061(AX8118-0210-0103 ) : B"}
	A_0062_AX8118_0210_0104 : AX8118_F7A82895;
	{attribute addProperty Name "A_0063(AX8206-0100-0101 )"}
	{attribute addProperty PreviousPort "A_0062(AX8118-0210-0104 ) : B"}
	A_0063_AX8206_0100_0101 : AX8206_63F473B4;
	{attribute addProperty Name "A_0064(AX8206-0100-0102 )"}
	{attribute addProperty PreviousPort "A_0063(AX8206-0100-0101 ) : B"}
	A_0064_AX8206_0100_0102 : AX8206_FA9FF81E;
	{attribute addProperty Name "A_0065(AX8206-0100-0103 )"}
	{attribute addProperty PreviousPort "A_0064(AX8206-0100-0102 ) : B"}
	A_0065_AX8206_0100_0103 : AX8206_FA9FF81E;
	{attribute addProperty Name "A_0066(AX8206-0100-0104 )"}
	{attribute addProperty PreviousPort "A_0065(AX8206-0100-0103 ) : B"}
	A_0066_AX8206_0100_0104 : AX8206_FA9FF81E;
	{attribute addProperty Name "A_0067(AX8206-0110-0102 )"}
	{attribute addProperty PreviousPort "A_0066(AX8206-0100-0104 ) : B"}
	A_0067_AX8206_0110_0102 : AX8206_FA9FF81E;
	{attribute addProperty Name "A_0068(AX8206-0110-0103 )"}
	{attribute addProperty PreviousPort "A_0067(AX8206-0110-0102 ) : B"}
	A_0068_AX8206_0110_0103 : AX8206_FA9FF81E;
	{attribute addProperty Name "A_0069(AX8206-0110-0104 )"}
	{attribute addProperty PreviousPort "A_0068(AX8206-0110-0103 ) : B"}
	A_0069_AX8206_0110_0104 : AX8206_FA9FF81E;
	{attribute addProperty Name "A_0070(AX8206-0200-0103 )"}
	{attribute addProperty PreviousPort "A_0069(AX8206-0110-0104 ) : B"}
	A_0070_AX8206_0200_0103 : AX8206_FA9FF81E;
	{attribute addProperty Name "A_0071(AX8206-0200-0104 )"}
	{attribute addProperty PreviousPort "A_0070(AX8206-0200-0103 ) : B"}
	A_0071_AX8206_0200_0104 : AX8206_FA9FF81E;
	{attribute addProperty Name "A_0072(AX8206-0210-0103 )"}
	{attribute addProperty PreviousPort "A_0071(AX8206-0200-0104 ) : B"}
	A_0072_AX8206_0210_0103 : AX8206_FA9FF81E;
	{attribute addProperty Name "A_0073(AX8206-0210-0104 )"}
	{attribute addProperty PreviousPort "A_0072(AX8206-0210-0103 ) : B"}
	A_0073_AX8206_0210_0104 : AX8206_FA9FF81E;
	{attribute addProperty Name "A_0074(EM7004-0000-9995)"}
	{attribute addProperty PreviousPort "A_0073(AX8206-0210-0104 ) : B"}
	A_0074_EM7004_0000_9995 : EM7004_866015E1;
	{attribute addProperty Name "A_0075(AX8118-0100-0101)"}
	{attribute addProperty PreviousPort "A_0074(EM7004-0000-9995) : B"}
	A_0075_AX8118_0100_0101 : AX8118_8297A621;
END_STRUCT
END_TYPE

// ---- DUTs/IO/Topology/EtherCAT_Master_Duplicates_CB89F35C.TcDUT
{attribute 'GeneratedUsingTerminal: IODEVICETYPE_ETHERCATPROT'}
{attribute addProperty BoxType "IODEVICETYPE_ETHERCATPROT"}
{attribute addProperty Id "boxesboxes_178979725785A_0076_AMP8000_0030_0103AMP8000_F7A82895113SyncUnitsSyncUnits_99E584AF18InputsInputs_25A0042B160OutputsOutputs_2397A10E106InfoDataInfoData_E68C61CD28"}
{attribute addProperty CRC "3414815580"}
{attribute addProperty Size "6210"}
{attribute addProperty Name "EtherCAT Master Duplicates"}
TYPE EtherCAT_Master_Duplicates_CB89F35C EXTENDS EtcMasterBase_62654B43 :
STRUCT
	{attribute addProperty Name "boxes"}
	{attribute addProperty PreviousPort "EtherCAT Master Duplicates : Master"}
	boxes : boxes_17897972;
	{attribute addProperty Name "A_0076(AMP8000-0030-0103)"}
	{attribute addProperty PreviousPort "boxes : C"}
	A_0076_AMP8000_0030_0103 : AMP8000_F7A82895;
	{attribute addProperty Name "SyncUnits"}
	SyncUnits : SyncUnits_99E584AF;
	{attribute addProperty Name "Inputs"}
	Inputs : Inputs_25A0042B;
	{attribute addProperty Name "Outputs"}
	Outputs : Outputs_2397A10E;
	{attribute addProperty Name "InfoData"}
	InfoData : InfoData_E68C61CD;
END_STRUCT
END_TYPE

// ---- DUTs/IO/Base/EtcSlaveBase_82538BE2.TcDUT

TYPE EtcSlaveBase_82538BE2 :
STRUCT
END_STRUCT
END_TYPE

// ---- DUTs/IO/Base/EtcSlaveBase_82538BE2.TcDUT

TYPE EtcSlaveBase_82538BE2 :
STRUCT
END_STRUCT
END_TYPE

// ---- DUTs/IO/Base/EtcSlaveBase_82538BE2.TcDUT

TYPE EtcSlaveBase_82538BE2 :
STRUCT
END_STRUCT
END_TYPE

// ---- DUTs/IO/Base/EtcSlaveTerminalBase_947E5A46.TcDUT

{attribute clr[Container(Layout.Stack)]}
{attribute clr[Group(Layout.GroupBox)]}
{attribute addProperty PreviousPort "Unknown"}
TYPE EtcSlaveTerminalBase_947E5A46 EXTENDS EtcSlaveBase_82538BE2 :
STRUCT
END_STRUCT
END_TYPE

// ---- DUTs/IO/Base/EtcSlaveBoxBase_77A0E4A7.TcDUT

{attribute clr[Container(Layout.Stack)]}
{attribute clr[Group(Layout.GroupBox)]}
{attribute addProperty PreviousPort "Unknown"}
TYPE EtcSlaveBoxBase_77A0E4A7 EXTENDS EtcSlaveBase_82538BE2 :
STRUCT
END_STRUCT
END_TYPE

// ---- DUTs/IO/Base/EtcSlaveEndTerminalBase_866C7F0C.TcDUT

{attribute clr[Container(Layout.Stack)]}
{attribute clr[Group(Layout.GroupBox)]}
{attribute addProperty PreviousPort "Unknown"}
TYPE EtcSlaveEndTerminalBase_866C7F0C EXTENDS EtcSlaveBase_82538BE2 :
STRUCT
END_STRUCT
END_TYPE

// ---- DUTs/IO/Base/InputBase_8311D824.TcDUT

TYPE InputBase_8311D824 :
STRUCT
END_STRUCT
END_TYPE

// ---- DUTs/IO/Base/OutputBase_10CEE7DE.TcDUT

TYPE OutputBase_10CEE7DE :
STRUCT
END_STRUCT
END_TYPE

// ---- DUTs/IO/Base/EtcMasterBase_62654B43.TcDUT

TYPE EtcMasterBase_62654B43 :
STRUCT
END_STRUCT
END_TYPE

// ---- GVLs/GVL_iXlinker.TcGVL
{attribute 'qualified_only'}
VAR_GLOBAL
		EtherCAT_Master_Duplicates : EtherCAT_Master_Duplicates_CB89F35C;
END_VAR

// ---- POUs/MAIN.TcPOU
PROGRAM MAIN
VAR
END_VAR

END_PROGRAM
